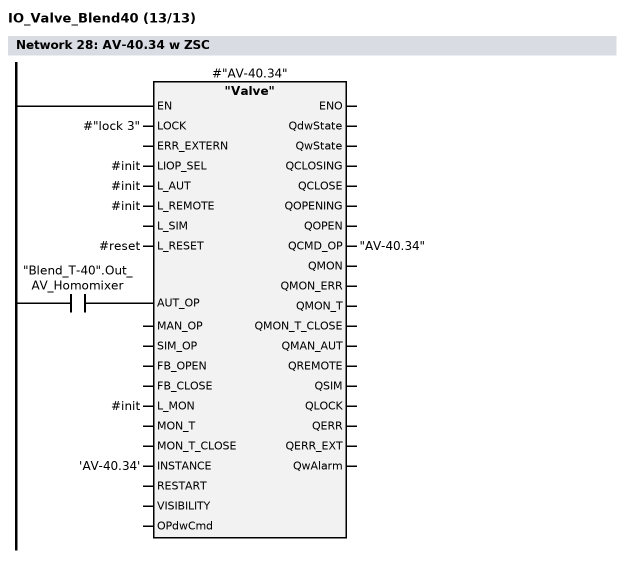
   RUNG wire#powerrail
      #"AV-40.34"(AUT_OP := wire#w1, LOCK := #"lock 3", ERR_EXTERN :=, LIOP_SEL := #init, L_AUT := #init, L_REMOTE := #init, L_SIM :=, L_RESET := #reset, MAN_OP :=, SIM_OP :=, FB_OPEN :=, FB_CLOSE :=, L_MON := #init, MON_T :=, MON_T_CLOSE :=, INSTANCE := 'AV-40.34', RESTART :=, VISIBILITY :=, OPdwCmd :=, QdwState =>, QwState =>, QCLOSING =>, QCLOSE =>, QOPENING =>, QOPEN =>, QCMD_OP => "AV-40.34", QMON =>, QMON_ERR =>, QMON_T =>, QMON_T_CLOSE =>, QMAN_AUT =>, QREMOTE =>, QSIM =>, QLOCK =>, QERR =>, QERR_EXT =>, QwAlarm =>)
   END_RUNG
   RUNG wire#powerrail
      Contact( "Blend_T-40".Out_AV_Homomixer )
   END_RUNG wire#w1
   // the same network as SCL:
   #"AV-40.34"(LOCK := #"lock 3",   // "Valve"
               LIOP_SEL := #init,
               L_AUT := #init,
               L_REMOTE := #init,
               L_RESET := #reset,
               AUT_OP := "Blend_T-40".Out_AV_Homomixer,
               L_MON := #init,
               INSTANCE := 'AV-40.34',
               QCMD_OP => "AV-40.34");
END_REGION
END_FUNCTION_BLOCK

FUNCTION_BLOCK "IO_Valve_Blend41"   // FB29, LAD
{ S7_Optimized_Access := 'FALSE' }
VERSION : 0.1
// stored: AutoNumber true, IsIECCheckEnabled false, SetENOAutomatically false, UDAEnableTagReadback false
   VAR_INPUT
      "lock 1" : Bool;
      "lock 2" : Bool;
      "lock 3" : Bool;
      "lock 4" : Bool;
      init : Bool;
      reset : Bool;
      testing : Bool;
   END_VAR
   VAR
      "AV-41.01" : "Valve";
      "AV-41.02" : "Valve";
      "AV-41.03" : "Valve";
      "AV-41.04" : "Valve";
      "AV-41.05" : "Valve";
      "AV-41.06" : "Valve";
      "AV-41.07" : "Valve";
      "AV-41.08" : "Valve";
      "AV-41.09" : "Valve";
      "AV-41.10" : "Valve";
      "AV-41.11" : "Valve";
      "AV-41.12" : "Valve";
      "AV-41.13" : "Valve";
      "AV-41.14" : "Valve";
      "AV-41.15" : "Valve";
      "AV-41.16" : "Valve";
      "AV-41.17" : "Valve";
      "AV-41.18" : "Valve";
      "AV-41.19" : "Valve";
      "AV-41.20" : "Valve";
      "AV-41.21" : "Valve";
      "AV-41.22" : "Valve";
      "AV-41.23" : "Valve";
      "AV-41.24" : "Valve";
      "AV-41.25" : "Valve";
      "AV-41.26" : "Valve";
      "AV-41.27" : "Valve";
      "AV-41.28" : "Valve";
      "AV-41.29" : "Valve";
      "AV-41.30" : "Valve";
      "AV-41.31" : "Valve";
      "AV-41.32" : "Valve";
      "AV-41.33" : "Valve";
      "AV-41.34" : "Valve";
   END_VAR
BEGIN

REGION Network 2 (SCL): FB OPEN AND CLOSE VALVE T-41
   IF #testing THEN
       // Statement section IF
       #"AV-41.01".FB_OPEN := #"AV-41.01".QCMD_OP;
       #"AV-41.01".FB_CLOSE := NOT #"AV-41.01".QCMD_OP;
       #"AV-41.02".FB_OPEN := #"AV-41.02".QCMD_OP;
       #"AV-41.02".FB_CLOSE := NOT #"AV-41.02".QCMD_OP;
       #"AV-41.03".FB_OPEN := #"AV-41.03".QCMD_OP;
       #"AV-41.03".FB_CLOSE := NOT #"AV-41.03".QCMD_OP;
       #"AV-41.04".FB_OPEN := #"AV-41.04".QCMD_OP;
       #"AV-41.04".FB_CLOSE := NOT #"AV-41.04".QCMD_OP;
       #"AV-41.05".FB_OPEN := #"AV-41.05".QCMD_OP;
       #"AV-41.05".FB_CLOSE := NOT #"AV-41.05".QCMD_OP;
       #"AV-41.06".FB_OPEN := #"AV-41.06".QCMD_OP;
       #"AV-41.06".FB_CLOSE := NOT #"AV-41.06".QCMD_OP;
       #"AV-41.07".FB_OPEN := #"AV-41.07".QCMD_OP;
       #"AV-41.07".FB_CLOSE := NOT #"AV-41.07".QCMD_OP;
       #"AV-41.08".FB_OPEN := #"AV-41.08".QCMD_OP;
       #"AV-41.08".FB_CLOSE := NOT #"AV-41.08".QCMD_OP;
       #"AV-41.09".FB_OPEN := #"AV-41.09".QCMD_OP;
       #"AV-41.09".FB_CLOSE := NOT #"AV-41.09".QCMD_OP;
       #"AV-41.10".FB_OPEN := #"AV-41.10".QCMD_OP;
       #"AV-41.10".FB_CLOSE := NOT #"AV-41.10".QCMD_OP;
       #"AV-41.11".FB_OPEN := #"AV-41.11".QCMD_OP;
       #"AV-41.11".FB_CLOSE := NOT #"AV-41.11".QCMD_OP;
       #"AV-41.12".FB_OPEN := #"AV-41.12".QCMD_OP;
       #"AV-41.12".FB_CLOSE := NOT #"AV-41.12".QCMD_OP;
       #"AV-41.13".FB_OPEN := #"AV-41.13".QCMD_OP;
       #"AV-41.13".FB_CLOSE := NOT #"AV-41.13".QCMD_OP;
       #"AV-41.14".FB_OPEN := #"AV-41.14".QCMD_OP;
       #"AV-41.14".FB_CLOSE := NOT #"AV-41.14".QCMD_OP;
       #"AV-41.15".FB_OPEN := #"AV-41.15".QCMD_OP;
       #"AV-41.15".FB_CLOSE := NOT #"AV-41.15".QCMD_OP;
       #"AV-41.16".FB_OPEN := #"AV-41.16".QCMD_OP;
       #"AV-41.16".FB_CLOSE := NOT #"AV-41.16".QCMD_OP;
       #"AV-41.17".FB_OPEN := #"AV-41.17".QCMD_OP;
       #"AV-41.17".FB_CLOSE := NOT #"AV-41.17".QCMD_OP;
       #"AV-41.18".FB_OPEN := #"AV-41.18".QCMD_OP;
       #"AV-41.18".FB_CLOSE := NOT #"AV-41.18".QCMD_OP;
       #"AV-41.19".FB_OPEN := #"AV-41.19".QCMD_OP;
       #"AV-41.19".FB_CLOSE := NOT #"AV-41.19".QCMD_OP;
       #"AV-41.20".FB_OPEN := #"AV-41.20".QCMD_OP;
       #"AV-41.20".FB_CLOSE := NOT #"AV-41.20".QCMD_OP;
       #"AV-41.21".FB_OPEN := #"AV-41.21".QCMD_OP;
       #"AV-41.21".FB_CLOSE := NOT #"AV-41.21".QCMD_OP;
       #"AV-41.22".FB_OPEN := #"AV-41.22".QCMD_OP;
       #"AV-41.22".FB_CLOSE := NOT #"AV-41.22".QCMD_OP;
       #"AV-41.23".FB_OPEN := #"AV-41.23".QCMD_OP;
       #"AV-41.23".FB_CLOSE := NOT #"AV-41.23".QCMD_OP;
       #"AV-41.24".FB_OPEN := #"AV-41.24".QCMD_OP;
       #"AV-41.24".FB_CLOSE := NOT #"AV-41.24".QCMD_OP;
       #"AV-41.25".FB_OPEN := #"AV-41.25".QCMD_OP;
       #"AV-41.25".FB_CLOSE := NOT #"AV-41.25".QCMD_OP;
       #"AV-41.26".FB_OPEN := #"AV-41.26".QCMD_OP;
       #"AV-41.26".FB_CLOSE := NOT #"AV-41.26".QCMD_OP;
       #"AV-41.27".FB_OPEN := #"AV-41.27".QCMD_OP;
       #"AV-41.27".FB_CLOSE := NOT #"AV-41.27".QCMD_OP;
       #"AV-41.28".FB_OPEN := #"AV-41.28".QCMD_OP;
       #"AV-41.28".FB_CLOSE := NOT #"AV-41.28".QCMD_OP;
       #"AV-41.29".FB_OPEN := #"AV-41.29".QCMD_OP;
       #"AV-41.29".FB_CLOSE := NOT #"AV-41.29".QCMD_OP;
       #"AV-41.30".FB_OPEN := #"AV-41.30".QCMD_OP;
       #"AV-41.30".FB_CLOSE := NOT #"AV-41.30".QCMD_OP;
       #"AV-41.31".FB_OPEN := #"AV-41.31".QCMD_OP;
       #"AV-41.31".FB_CLOSE := NOT #"AV-41.31".QCMD_OP;
       #"AV-41.32".FB_OPEN := #"AV-41.32".QCMD_OP;
       #"AV-41.32".FB_CLOSE := NOT #"AV-41.32".QCMD_OP;
       #"AV-41.33".FB_OPEN := #"AV-41.33".QCMD_OP;
       #"AV-41.33".FB_CLOSE := NOT #"AV-41.33".QCMD_OP;
       #"AV-41.34".FB_OPEN := #"AV-41.34".QCMD_OP;
       #"AV-41.34".FB_CLOSE := NOT #"AV-41.34".QCMD_OP;
   ELSE
       // Statement section ELSE
       #"AV-41.01".FB_OPEN := #"AV-41.01".QCMD_OP;
       #"AV-41.01".FB_CLOSE := NOT #"AV-41.01".QCMD_OP;
       #"AV-41.02".FB_OPEN := NOT "ZSC-41.02";
       #"AV-41.02".FB_CLOSE := "ZSC-41.02";
       #"AV-41.03".FB_OPEN := NOT "ZSC-41.03";
       #"AV-41.03".FB_CLOSE := "ZSC-41.03";
       #"AV-41.04".FB_OPEN := #"AV-41.04".QCMD_OP;
       #"AV-41.04".FB_CLOSE := NOT #"AV-41.04".QCMD_OP;
       #"AV-41.05".FB_OPEN := NOT "ZSC-41.05";
       #"AV-41.05".FB_CLOSE := "ZSC-41.05";
       #"AV-41.06".FB_OPEN := NOT "ZSC-41.06";
       #"AV-41.06".FB_CLOSE := "ZSC-41.06";
       #"AV-41.07".FB_OPEN := #"AV-41.07".QCMD_OP;
       #"AV-41.07".FB_CLOSE := NOT #"AV-41.07".QCMD_OP;
       #"AV-41.08".FB_OPEN := NOT "ZSC-41.08";
       #"AV-41.08".FB_CLOSE := "ZSC-41.08";
       #"AV-41.09".FB_OPEN := NOT "ZSC-41.09";
       #"AV-41.09".FB_CLOSE := "ZSC-41.09";
       #"AV-41.10".FB_OPEN := #"AV-41.10".QCMD_OP;
       #"AV-41.10".FB_CLOSE := NOT #"AV-41.10".QCMD_OP;
       #"AV-41.11".FB_OPEN := NOT "ZSC-41.11";
       #"AV-41.11".FB_CLOSE := "ZSC-41.11";
       #"AV-41.12".FB_OPEN := #"AV-41.12".QCMD_OP;
       #"AV-41.12".FB_CLOSE := NOT #"AV-41.12".QCMD_OP;
       #"AV-41.13".FB_OPEN := #"AV-41.13".QCMD_OP;
       #"AV-41.13".FB_CLOSE := NOT #"AV-41.13".QCMD_OP;
       #"AV-41.14".FB_OPEN := NOT "ZSC-41.14";
       #"AV-41.14".FB_CLOSE := "ZSC-41.14";
       #"AV-41.15".FB_OPEN := #"AV-41.15".QCMD_OP;
       #"AV-41.15".FB_CLOSE := NOT #"AV-41.15".QCMD_OP;
       #"AV-41.16".FB_OPEN := #"AV-41.16".QCMD_OP;
       #"AV-41.16".FB_CLOSE := NOT #"AV-41.16".QCMD_OP;
       #"AV-41.17".FB_OPEN := NOT "ZSC-41.17";
       #"AV-41.17".FB_CLOSE := "ZSC-41.17";
       #"AV-41.18".FB_OPEN := #"AV-41.18".QCMD_OP;
       #"AV-41.18".FB_CLOSE := NOT #"AV-41.18".QCMD_OP;
       #"AV-41.19".FB_OPEN := #"AV-41.19".QCMD_OP;
       #"AV-41.19".FB_CLOSE := NOT #"AV-41.19".QCMD_OP;
       #"AV-41.20".FB_OPEN := NOT "ZSC-41.20";
       #"AV-41.20".FB_CLOSE := "ZSC-41.20";
       #"AV-41.21".FB_OPEN := NOT "ZSC-41.21";
       #"AV-41.21".FB_CLOSE := "ZSC-41.21";
       #"AV-41.22".FB_OPEN := #"AV-41.22".QCMD_OP;
       #"AV-41.22".FB_CLOSE := NOT #"AV-41.22".QCMD_OP;
       #"AV-41.23".FB_OPEN := NOT "ZSC-41.23";
       #"AV-41.23".FB_CLOSE := "ZSC-41.23";
       #"AV-41.24".FB_OPEN := NOT "ZSC-41.24";
       #"AV-41.24".FB_CLOSE := "ZSC-41.24";
       #"AV-41.25".FB_OPEN := NOT "ZSC-41.25";
       #"AV-41.25".FB_CLOSE := "ZSC-41.25";
       #"AV-41.26".FB_OPEN := #"AV-41.26".QCMD_OP;
       #"AV-41.26".FB_CLOSE := NOT #"AV-41.26".QCMD_OP;
       #"AV-41.27".FB_OPEN := NOT "ZSC-41.27";
       #"AV-41.27".FB_CLOSE := "ZSC-41.27";
       #"AV-41.28".FB_OPEN := NOT "ZSC-41.28";
       #"AV-41.28".FB_CLOSE := "ZSC-41.28";
       #"AV-41.29".FB_OPEN := #"AV-41.29".QCMD_OP;
       #"AV-41.29".FB_CLOSE := NOT #"AV-41.29".QCMD_OP;
       #"AV-41.30".FB_OPEN := #"AV-41.30".QCMD_OP;
       #"AV-41.30".FB_CLOSE := NOT #"AV-41.30".QCMD_OP;
       #"AV-41.31".FB_OPEN := NOT "ZSC-41.31";
       #"AV-41.31".FB_CLOSE := "ZSC-41.31";
       #"AV-41.32".FB_OPEN := NOT "ZSC-41.32";
       #"AV-41.32".FB_CLOSE := "ZSC-41.32";
       #"AV-41.33".FB_OPEN := NOT "ZSC-41.33";
       #"AV-41.33".FB_CLOSE := "ZSC-41.33";
       #"AV-41.34".FB_OPEN := NOT "ZSC-41.34";
       #"AV-41.34".FB_CLOSE := "ZSC-41.34";
   END_IF;
END_REGION

NETWORK
TITLE = FB MONITORING TIME VALVE T-41
// FB OPEN TIME
      L     T#20s;
      T     #"AV-41.01".MON_T;
      T     #"AV-41.02".MON_T;
      T     #"AV-41.03".MON_T;
      T     #"AV-41.04".MON_T;
      T     #"AV-41.05".MON_T;
      T     #"AV-41.06".MON_T;
      T     #"AV-41.07".MON_T;
      T     #"AV-41.08".MON_T;
      T     #"AV-41.09".MON_T;
      T     #"AV-41.10".MON_T;
      T     #"AV-41.11".MON_T;
      T     #"AV-41.12".MON_T;
      T     #"AV-41.13".MON_T;
      T     #"AV-41.14".MON_T;
      T     #"AV-41.15".MON_T;
      T     #"AV-41.16".MON_T;
      T     #"AV-41.17".MON_T;
      T     #"AV-41.18".MON_T;
      T     #"AV-41.19".MON_T;
      T     #"AV-41.20".MON_T;
      T     #"AV-41.21".MON_T;
      T     #"AV-41.22".MON_T;
      T     #"AV-41.23".MON_T;
      T     #"AV-41.24".MON_T;
      T     #"AV-41.25".MON_T;
      T     #"AV-41.26".MON_T;
      T     #"AV-41.27".MON_T;
      T     #"AV-41.28".MON_T;
      T     #"AV-41.29".MON_T;
      T     #"AV-41.30".MON_T;
      T     #"AV-41.31".MON_T;
      T     #"AV-41.32".MON_T;
      T     #"AV-41.33".MON_T;
      T     #"AV-41.34".MON_T;
// FB CLOSE TIME
      L     T#20s;
      T     #"AV-41.01".MON_T_CLOSE;
      T     #"AV-41.02".MON_T_CLOSE;
      T     #"AV-41.03".MON_T_CLOSE;
      T     #"AV-41.04".MON_T_CLOSE;
      T     #"AV-41.05".MON_T_CLOSE;
      T     #"AV-41.06".MON_T_CLOSE;
      T     #"AV-41.07".MON_T_CLOSE;
      T     #"AV-41.08".MON_T_CLOSE;
      T     #"AV-41.09".MON_T_CLOSE;
      T     #"AV-41.10".MON_T_CLOSE;
      T     #"AV-41.11".MON_T_CLOSE;
      T     #"AV-41.12".MON_T_CLOSE;
      T     #"AV-41.13".MON_T_CLOSE;
      T     #"AV-41.14".MON_T_CLOSE;
      T     #"AV-41.15".MON_T_CLOSE;
      T     #"AV-41.16".MON_T_CLOSE;
      T     #"AV-41.17".MON_T_CLOSE;
      T     #"AV-41.18".MON_T_CLOSE;
      T     #"AV-41.19".MON_T_CLOSE;
      T     #"AV-41.20".MON_T_CLOSE;
      T     #"AV-41.21".MON_T_CLOSE;
      T     #"AV-41.22".MON_T_CLOSE;
      T     #"AV-41.23".MON_T_CLOSE;
      T     #"AV-41.24".MON_T_CLOSE;
      T     #"AV-41.25".MON_T_CLOSE;
      T     #"AV-41.26".MON_T_CLOSE;
      T     #"AV-41.27".MON_T_CLOSE;
      T     #"AV-41.28".MON_T_CLOSE;
      T     #"AV-41.29".MON_T_CLOSE;
      T     #"AV-41.30".MON_T_CLOSE;
      T     #"AV-41.31".MON_T_CLOSE;
      T     #"AV-41.32".MON_T_CLOSE;
      T     #"AV-41.33".MON_T_CLOSE;
      T     #"AV-41.34".MON_T_CLOSE;

REGION Network 4: AV-41.01
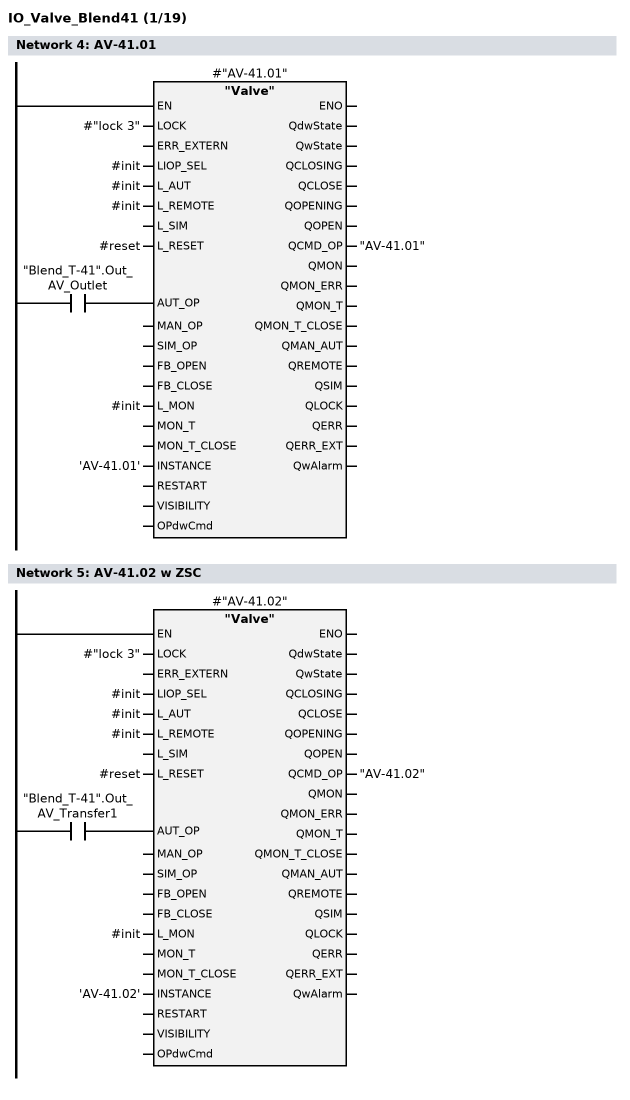
   RUNG wire#powerrail
      #"AV-41.01"(AUT_OP := wire#w1, LOCK := #"lock 3", ERR_EXTERN :=, LIOP_SEL := #init, L_AUT := #init, L_REMOTE := #init, L_SIM :=, L_RESET := #reset, MAN_OP :=, SIM_OP :=, FB_OPEN :=, FB_CLOSE :=, L_MON := #init, MON_T :=, MON_T_CLOSE :=, INSTANCE := 'AV-41.01', RESTART :=, VISIBILITY :=, OPdwCmd :=, QdwState =>, QwState =>, QCLOSING =>, QCLOSE =>, QOPENING =>, QOPEN =>, QCMD_OP => "AV-41.01", QMON =>, QMON_ERR =>, QMON_T =>, QMON_T_CLOSE =>, QMAN_AUT =>, QREMOTE =>, QSIM =>, QLOCK =>, QERR =>, QERR_EXT =>, QwAlarm =>)
   END_RUNG
   RUNG wire#powerrail
      Contact( "Blend_T-41".Out_AV_Outlet )
   END_RUNG wire#w1
   // the same network as SCL:
   #"AV-41.01"(LOCK := #"lock 3",   // "Valve"
               LIOP_SEL := #init,
               L_AUT := #init,
               L_REMOTE := #init,
               L_RESET := #reset,
               AUT_OP := "Blend_T-41".Out_AV_Outlet,
               L_MON := #init,
               INSTANCE := 'AV-41.01',
               QCMD_OP => "AV-41.01");
END_REGION

REGION Network 5: AV-41.02 w ZSC
   RUNG wire#powerrail
      #"AV-41.02"(AUT_OP := wire#w1, LOCK := #"lock 3", ERR_EXTERN :=, LIOP_SEL := #init, L_AUT := #init, L_REMOTE := #init, L_SIM :=, L_RESET := #reset, MAN_OP :=, SIM_OP :=, FB_OPEN :=, FB_CLOSE :=, L_MON := #init, MON_T :=, MON_T_CLOSE :=, INSTANCE := 'AV-41.02', RESTART :=, VISIBILITY :=, OPdwCmd :=, QdwState =>, QwState =>, QCLOSING =>, QCLOSE =>, QOPENING =>, QOPEN =>, QCMD_OP => "AV-41.02", QMON =>, QMON_ERR =>, QMON_T =>, QMON_T_CLOSE =>, QMAN_AUT =>, QREMOTE =>, QSIM =>, QLOCK =>, QERR =>, QERR_EXT =>, QwAlarm =>)
   END_RUNG
   RUNG wire#powerrail
      Contact( "Blend_T-41".Out_AV_Transfer1 )
   END_RUNG wire#w1
   // the same network as SCL:
   #"AV-41.02"(LOCK := #"lock 3",   // "Valve"
               LIOP_SEL := #init,
               L_AUT := #init,
               L_REMOTE := #init,
               L_RESET := #reset,
               AUT_OP := "Blend_T-41".Out_AV_Transfer1,
               L_MON := #init,
               INSTANCE := 'AV-41.02',
               QCMD_OP => "AV-41.02");
END_REGION

REGION Network 6: AV-41.03 w ZSC
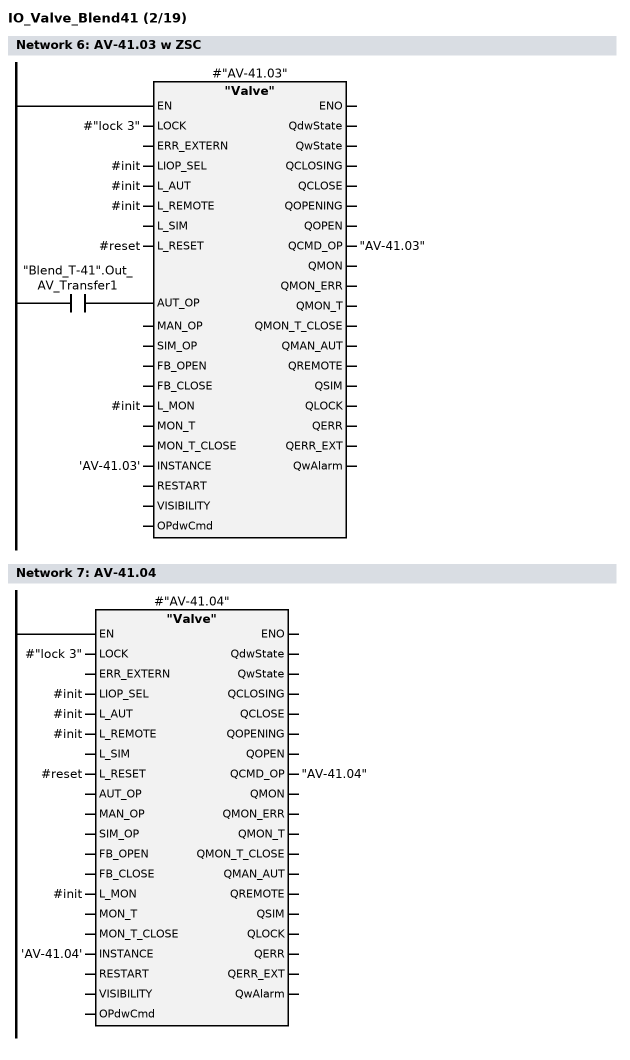
   RUNG wire#powerrail
      #"AV-41.03"(AUT_OP := wire#w1, LOCK := #"lock 3", ERR_EXTERN :=, LIOP_SEL := #init, L_AUT := #init, L_REMOTE := #init, L_SIM :=, L_RESET := #reset, MAN_OP :=, SIM_OP :=, FB_OPEN :=, FB_CLOSE :=, L_MON := #init, MON_T :=, MON_T_CLOSE :=, INSTANCE := 'AV-41.03', RESTART :=, VISIBILITY :=, OPdwCmd :=, QdwState =>, QwState =>, QCLOSING =>, QCLOSE =>, QOPENING =>, QOPEN =>, QCMD_OP => "AV-41.03", QMON =>, QMON_ERR =>, QMON_T =>, QMON_T_CLOSE =>, QMAN_AUT =>, QREMOTE =>, QSIM =>, QLOCK =>, QERR =>, QERR_EXT =>, QwAlarm =>)
   END_RUNG
   RUNG wire#powerrail
      Contact( "Blend_T-41".Out_AV_Transfer1 )
   END_RUNG wire#w1
   // the same network as SCL:
   #"AV-41.03"(LOCK := #"lock 3",   // "Valve"
               LIOP_SEL := #init,
               L_AUT := #init,
               L_REMOTE := #init,
               L_RESET := #reset,
               AUT_OP := "Blend_T-41".Out_AV_Transfer1,
               L_MON := #init,
               INSTANCE := 'AV-41.03',
               QCMD_OP => "AV-41.03");
END_REGION

REGION Network 7: AV-41.04
   RUNG wire#powerrail
      #"AV-41.04"(LOCK := #"lock 3", ERR_EXTERN :=, LIOP_SEL := #init, L_AUT := #init, L_REMOTE := #init, L_SIM :=, L_RESET := #reset, AUT_OP :=, MAN_OP :=, SIM_OP :=, FB_OPEN :=, FB_CLOSE :=, L_MON := #init, MON_T :=, MON_T_CLOSE :=, INSTANCE := 'AV-41.04', RESTART :=, VISIBILITY :=, OPdwCmd :=, QdwState =>, QwState =>, QCLOSING =>, QCLOSE =>, QOPENING =>, QOPEN =>, QCMD_OP => "AV-41.04", QMON =>, QMON_ERR =>, QMON_T =>, QMON_T_CLOSE =>, QMAN_AUT =>, QREMOTE =>, QSIM =>, QLOCK =>, QERR =>, QERR_EXT =>, QwAlarm =>)
   END_RUNG
   // the same network as SCL:
   #"AV-41.04"(LOCK := #"lock 3",   // "Valve"
               LIOP_SEL := #init,
               L_AUT := #init,
               L_REMOTE := #init,
               L_RESET := #reset,
               L_MON := #init,
               INSTANCE := 'AV-41.04',
               QCMD_OP => "AV-41.04");
END_REGION

REGION Network 8: AV-41.05 w ZSC
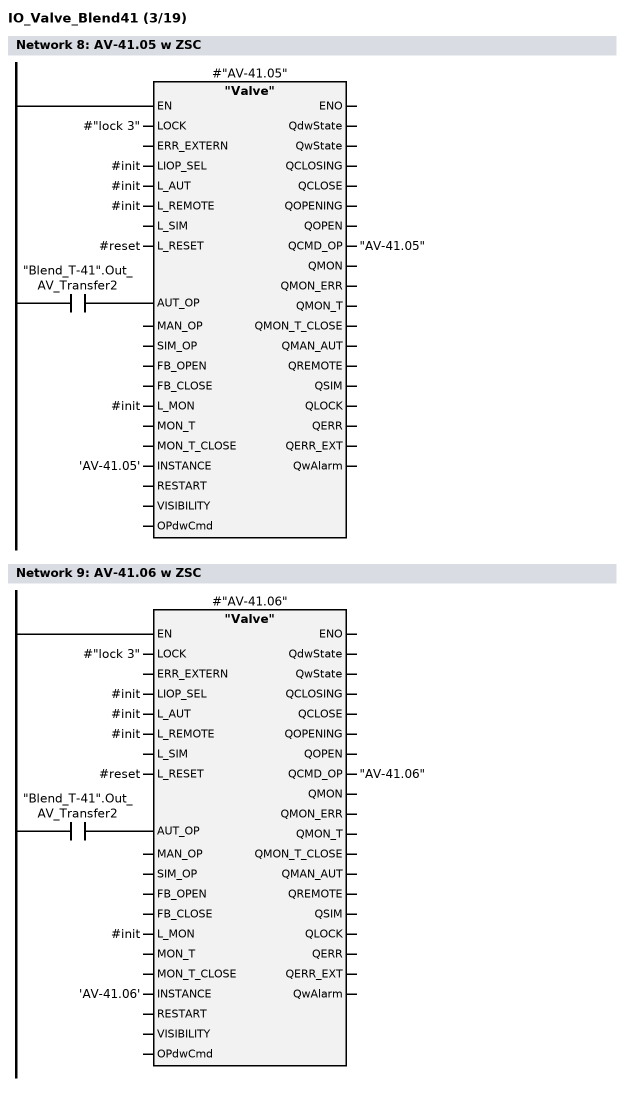
   RUNG wire#powerrail
      #"AV-41.05"(AUT_OP := wire#w1, LOCK := #"lock 3", ERR_EXTERN :=, LIOP_SEL := #init, L_AUT := #init, L_REMOTE := #init, L_SIM :=, L_RESET := #reset, MAN_OP :=, SIM_OP :=, FB_OPEN :=, FB_CLOSE :=, L_MON := #init, MON_T :=, MON_T_CLOSE :=, INSTANCE := 'AV-41.05', RESTART :=, VISIBILITY :=, OPdwCmd :=, QdwState =>, QwState =>, QCLOSING =>, QCLOSE =>, QOPENING =>, QOPEN =>, QCMD_OP => "AV-41.05", QMON =>, QMON_ERR =>, QMON_T =>, QMON_T_CLOSE =>, QMAN_AUT =>, QREMOTE =>, QSIM =>, QLOCK =>, QERR =>, QERR_EXT =>, QwAlarm =>)
   END_RUNG
   RUNG wire#powerrail
      Contact( "Blend_T-41".Out_AV_Transfer2 )
   END_RUNG wire#w1
   // the same network as SCL:
   #"AV-41.05"(LOCK := #"lock 3",   // "Valve"
               LIOP_SEL := #init,
               L_AUT := #init,
               L_REMOTE := #init,
               L_RESET := #reset,
               AUT_OP := "Blend_T-41".Out_AV_Transfer2,
               L_MON := #init,
               INSTANCE := 'AV-41.05',
               QCMD_OP => "AV-41.05");
END_REGION

REGION Network 9: AV-41.06 w ZSC
   RUNG wire#powerrail
      #"AV-41.06"(AUT_OP := wire#w1, LOCK := #"lock 3", ERR_EXTERN :=, LIOP_SEL := #init, L_AUT := #init, L_REMOTE := #init, L_SIM :=, L_RESET := #reset, MAN_OP :=, SIM_OP :=, FB_OPEN :=, FB_CLOSE :=, L_MON := #init, MON_T :=, MON_T_CLOSE :=, INSTANCE := 'AV-41.06', RESTART :=, VISIBILITY :=, OPdwCmd :=, QdwState =>, QwState =>, QCLOSING =>, QCLOSE =>, QOPENING =>, QOPEN =>, QCMD_OP => "AV-41.06", QMON =>, QMON_ERR =>, QMON_T =>, QMON_T_CLOSE =>, QMAN_AUT =>, QREMOTE =>, QSIM =>, QLOCK =>, QERR =>, QERR_EXT =>, QwAlarm =>)
   END_RUNG
   RUNG wire#powerrail
      Contact( "Blend_T-41".Out_AV_Transfer2 )
   END_RUNG wire#w1
   // the same network as SCL:
   #"AV-41.06"(LOCK := #"lock 3",   // "Valve"
               LIOP_SEL := #init,
               L_AUT := #init,
               L_REMOTE := #init,
               L_RESET := #reset,
               AUT_OP := "Blend_T-41".Out_AV_Transfer2,
               L_MON := #init,
               INSTANCE := 'AV-41.06',
               QCMD_OP => "AV-41.06");
END_REGION

REGION Network 10: AV-41.07
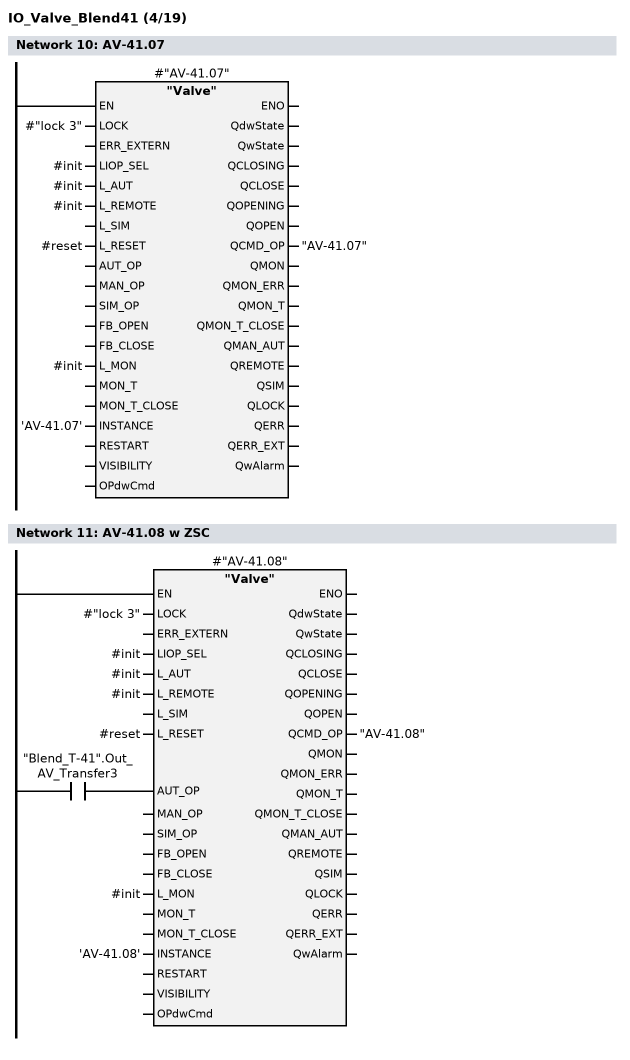
   RUNG wire#powerrail
      #"AV-41.07"(LOCK := #"lock 3", ERR_EXTERN :=, LIOP_SEL := #init, L_AUT := #init, L_REMOTE := #init, L_SIM :=, L_RESET := #reset, AUT_OP :=, MAN_OP :=, SIM_OP :=, FB_OPEN :=, FB_CLOSE :=, L_MON := #init, MON_T :=, MON_T_CLOSE :=, INSTANCE := 'AV-41.07', RESTART :=, VISIBILITY :=, OPdwCmd :=, QdwState =>, QwState =>, QCLOSING =>, QCLOSE =>, QOPENING =>, QOPEN =>, QCMD_OP => "AV-41.07", QMON =>, QMON_ERR =>, QMON_T =>, QMON_T_CLOSE =>, QMAN_AUT =>, QREMOTE =>, QSIM =>, QLOCK =>, QERR =>, QERR_EXT =>, QwAlarm =>)
   END_RUNG
   // the same network as SCL:
   #"AV-41.07"(LOCK := #"lock 3",   // "Valve"
               LIOP_SEL := #init,
               L_AUT := #init,
               L_REMOTE := #init,
               L_RESET := #reset,
               L_MON := #init,
               INSTANCE := 'AV-41.07',
               QCMD_OP => "AV-41.07");
END_REGION

REGION Network 11: AV-41.08 w ZSC
   RUNG wire#powerrail
      #"AV-41.08"(AUT_OP := wire#w1, LOCK := #"lock 3", ERR_EXTERN :=, LIOP_SEL := #init, L_AUT := #init, L_REMOTE := #init, L_SIM :=, L_RESET := #reset, MAN_OP :=, SIM_OP :=, FB_OPEN :=, FB_CLOSE :=, L_MON := #init, MON_T :=, MON_T_CLOSE :=, INSTANCE := 'AV-41.08', RESTART :=, VISIBILITY :=, OPdwCmd :=, QdwState =>, QwState =>, QCLOSING =>, QCLOSE =>, QOPENING =>, QOPEN =>, QCMD_OP => "AV-41.08", QMON =>, QMON_ERR =>, QMON_T =>, QMON_T_CLOSE =>, QMAN_AUT =>, QREMOTE =>, QSIM =>, QLOCK =>, QERR =>, QERR_EXT =>, QwAlarm =>)
   END_RUNG
   RUNG wire#powerrail
      Contact( "Blend_T-41".Out_AV_Transfer3 )
   END_RUNG wire#w1
   // the same network as SCL:
   #"AV-41.08"(LOCK := #"lock 3",   // "Valve"
               LIOP_SEL := #init,
               L_AUT := #init,
               L_REMOTE := #init,
               L_RESET := #reset,
               AUT_OP := "Blend_T-41".Out_AV_Transfer3,
               L_MON := #init,
               INSTANCE := 'AV-41.08',
               QCMD_OP => "AV-41.08");
END_REGION

REGION Network 12: AV-41.09 w ZSC
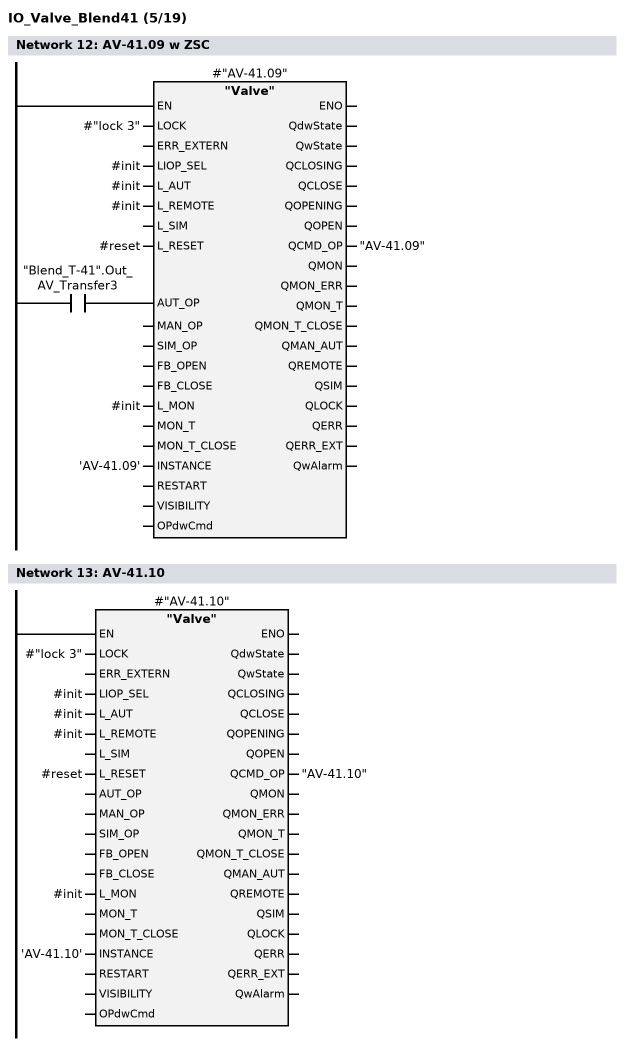
   RUNG wire#powerrail
      #"AV-41.09"(AUT_OP := wire#w1, LOCK := #"lock 3", ERR_EXTERN :=, LIOP_SEL := #init, L_AUT := #init, L_REMOTE := #init, L_SIM :=, L_RESET := #reset, MAN_OP :=, SIM_OP :=, FB_OPEN :=, FB_CLOSE :=, L_MON := #init, MON_T :=, MON_T_CLOSE :=, INSTANCE := 'AV-41.09', RESTART :=, VISIBILITY :=, OPdwCmd :=, QdwState =>, QwState =>, QCLOSING =>, QCLOSE =>, QOPENING =>, QOPEN =>, QCMD_OP => "AV-41.09", QMON =>, QMON_ERR =>, QMON_T =>, QMON_T_CLOSE =>, QMAN_AUT =>, QREMOTE =>, QSIM =>, QLOCK =>, QERR =>, QERR_EXT =>, QwAlarm =>)
   END_RUNG
   RUNG wire#powerrail
      Contact( "Blend_T-41".Out_AV_Transfer3 )
   END_RUNG wire#w1
   // the same network as SCL:
   #"AV-41.09"(LOCK := #"lock 3",   // "Valve"
               LIOP_SEL := #init,
               L_AUT := #init,
               L_REMOTE := #init,
               L_RESET := #reset,
               AUT_OP := "Blend_T-41".Out_AV_Transfer3,
               L_MON := #init,
               INSTANCE := 'AV-41.09',
               QCMD_OP => "AV-41.09");
END_REGION

REGION Network 13: AV-41.10
   RUNG wire#powerrail
      #"AV-41.10"(LOCK := #"lock 3", ERR_EXTERN :=, LIOP_SEL := #init, L_AUT := #init, L_REMOTE := #init, L_SIM :=, L_RESET := #reset, AUT_OP :=, MAN_OP :=, SIM_OP :=, FB_OPEN :=, FB_CLOSE :=, L_MON := #init, MON_T :=, MON_T_CLOSE :=, INSTANCE := 'AV-41.10', RESTART :=, VISIBILITY :=, OPdwCmd :=, QdwState =>, QwState =>, QCLOSING =>, QCLOSE =>, QOPENING =>, QOPEN =>, QCMD_OP => "AV-41.10", QMON =>, QMON_ERR =>, QMON_T =>, QMON_T_CLOSE =>, QMAN_AUT =>, QREMOTE =>, QSIM =>, QLOCK =>, QERR =>, QERR_EXT =>, QwAlarm =>)
   END_RUNG
   // the same network as SCL:
   #"AV-41.10"(LOCK := #"lock 3",   // "Valve"
               LIOP_SEL := #init,
               L_AUT := #init,
               L_REMOTE := #init,
               L_RESET := #reset,
               L_MON := #init,
               INSTANCE := 'AV-41.10',
               QCMD_OP => "AV-41.10");
END_REGION

REGION Network 14: AV-41.11 w ZSC
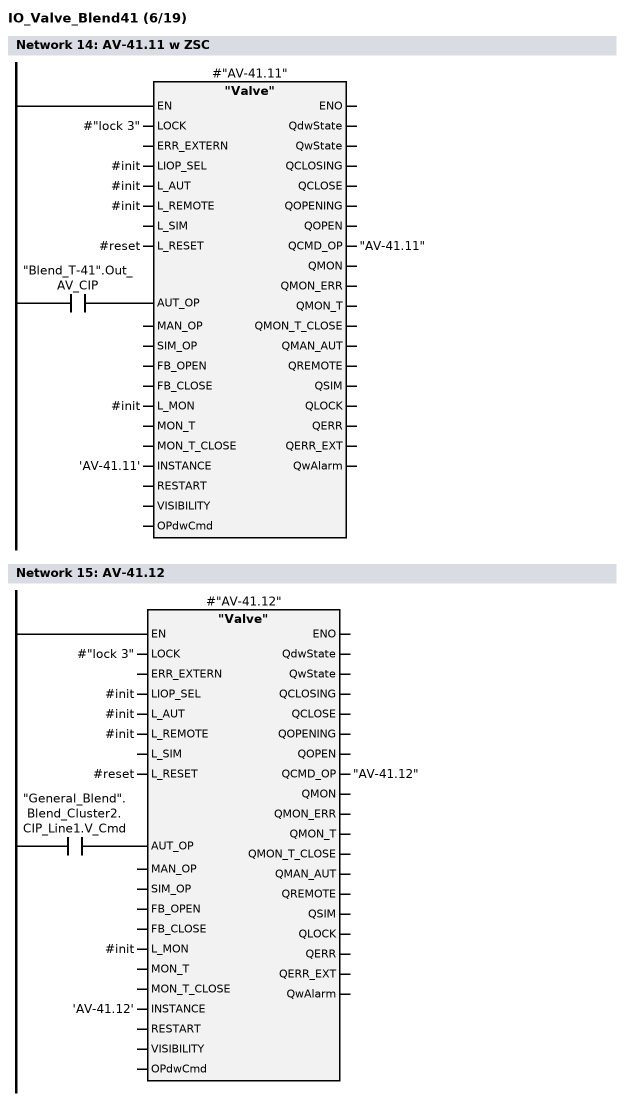
   RUNG wire#powerrail
      #"AV-41.11"(AUT_OP := wire#w1, LOCK := #"lock 3", ERR_EXTERN :=, LIOP_SEL := #init, L_AUT := #init, L_REMOTE := #init, L_SIM :=, L_RESET := #reset, MAN_OP :=, SIM_OP :=, FB_OPEN :=, FB_CLOSE :=, L_MON := #init, MON_T :=, MON_T_CLOSE :=, INSTANCE := 'AV-41.11', RESTART :=, VISIBILITY :=, OPdwCmd :=, QdwState =>, QwState =>, QCLOSING =>, QCLOSE =>, QOPENING =>, QOPEN =>, QCMD_OP => "AV-41.11", QMON =>, QMON_ERR =>, QMON_T =>, QMON_T_CLOSE =>, QMAN_AUT =>, QREMOTE =>, QSIM =>, QLOCK =>, QERR =>, QERR_EXT =>, QwAlarm =>)
   END_RUNG
   RUNG wire#powerrail
      Contact( "Blend_T-41".Out_AV_CIP )
   END_RUNG wire#w1
   // the same network as SCL:
   #"AV-41.11"(LOCK := #"lock 3",   // "Valve"
               LIOP_SEL := #init,
               L_AUT := #init,
               L_REMOTE := #init,
               L_RESET := #reset,
               AUT_OP := "Blend_T-41".Out_AV_CIP,
               L_MON := #init,
               INSTANCE := 'AV-41.11',
               QCMD_OP => "AV-41.11");
END_REGION

REGION Network 15: AV-41.12
   RUNG wire#powerrail
      #"AV-41.12"(AUT_OP := wire#w1, LOCK := #"lock 3", ERR_EXTERN :=, LIOP_SEL := #init, L_AUT := #init, L_REMOTE := #init, L_SIM :=, L_RESET := #reset, MAN_OP :=, SIM_OP :=, FB_OPEN :=, FB_CLOSE :=, L_MON := #init, MON_T :=, MON_T_CLOSE :=, INSTANCE := 'AV-41.12', RESTART :=, VISIBILITY :=, OPdwCmd :=, QdwState =>, QwState =>, QCLOSING =>, QCLOSE =>, QOPENING =>, QOPEN =>, QCMD_OP => "AV-41.12", QMON =>, QMON_ERR =>, QMON_T =>, QMON_T_CLOSE =>, QMAN_AUT =>, QREMOTE =>, QSIM =>, QLOCK =>, QERR =>, QERR_EXT =>, QwAlarm =>)
   END_RUNG
   RUNG wire#powerrail
      Contact( "General_Blend".Blend_Cluster2.CIP_Line1.V_Cmd )
   END_RUNG wire#w1
   // the same network as SCL:
   #"AV-41.12"(LOCK := #"lock 3",   // "Valve"
               LIOP_SEL := #init,
               L_AUT := #init,
               L_REMOTE := #init,
               L_RESET := #reset,
               AUT_OP := "General_Blend".Blend_Cluster2.CIP_Line1.V_Cmd,
               L_MON := #init,
               INSTANCE := 'AV-41.12',
               QCMD_OP => "AV-41.12");
END_REGION

REGION Network 16: AV-41.13
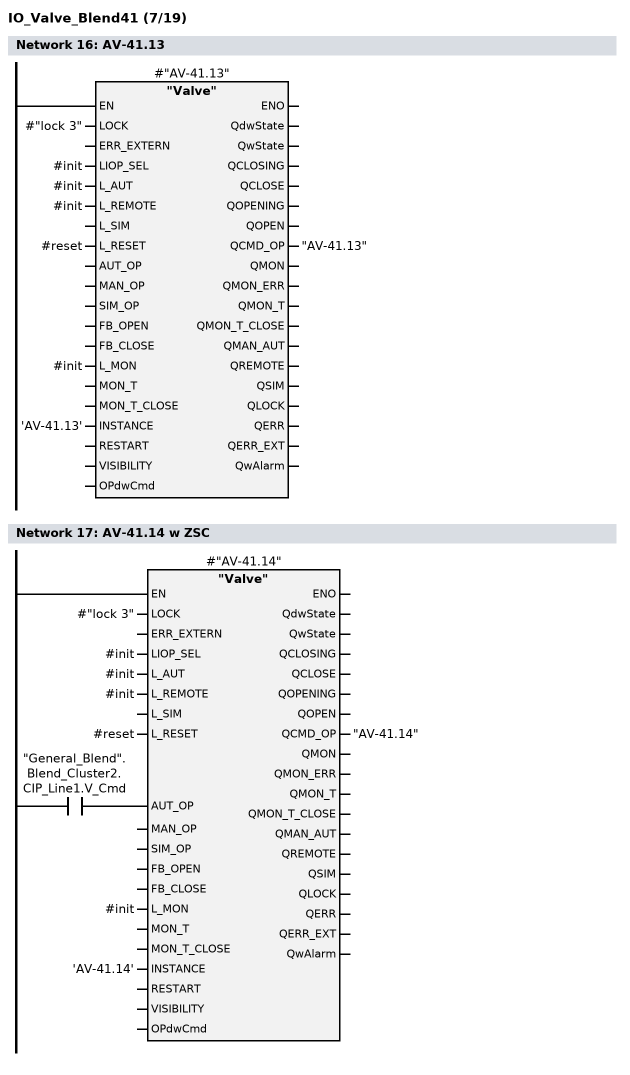
   RUNG wire#powerrail
      #"AV-41.13"(LOCK := #"lock 3", ERR_EXTERN :=, LIOP_SEL := #init, L_AUT := #init, L_REMOTE := #init, L_SIM :=, L_RESET := #reset, AUT_OP :=, MAN_OP :=, SIM_OP :=, FB_OPEN :=, FB_CLOSE :=, L_MON := #init, MON_T :=, MON_T_CLOSE :=, INSTANCE := 'AV-41.13', RESTART :=, VISIBILITY :=, OPdwCmd :=, QdwState =>, QwState =>, QCLOSING =>, QCLOSE =>, QOPENING =>, QOPEN =>, QCMD_OP => "AV-41.13", QMON =>, QMON_ERR =>, QMON_T =>, QMON_T_CLOSE =>, QMAN_AUT =>, QREMOTE =>, QSIM =>, QLOCK =>, QERR =>, QERR_EXT =>, QwAlarm =>)
   END_RUNG
   // the same network as SCL:
   #"AV-41.13"(LOCK := #"lock 3",   // "Valve"
               LIOP_SEL := #init,
               L_AUT := #init,
               L_REMOTE := #init,
               L_RESET := #reset,
               L_MON := #init,
               INSTANCE := 'AV-41.13',
               QCMD_OP => "AV-41.13");
END_REGION

REGION Network 17: AV-41.14 w ZSC
   RUNG wire#powerrail
      #"AV-41.14"(AUT_OP := wire#w1, LOCK := #"lock 3", ERR_EXTERN :=, LIOP_SEL := #init, L_AUT := #init, L_REMOTE := #init, L_SIM :=, L_RESET := #reset, MAN_OP :=, SIM_OP :=, FB_OPEN :=, FB_CLOSE :=, L_MON := #init, MON_T :=, MON_T_CLOSE :=, INSTANCE := 'AV-41.14', RESTART :=, VISIBILITY :=, OPdwCmd :=, QdwState =>, QwState =>, QCLOSING =>, QCLOSE =>, QOPENING =>, QOPEN =>, QCMD_OP => "AV-41.14", QMON =>, QMON_ERR =>, QMON_T =>, QMON_T_CLOSE =>, QMAN_AUT =>, QREMOTE =>, QSIM =>, QLOCK =>, QERR =>, QERR_EXT =>, QwAlarm =>)
   END_RUNG
   RUNG wire#powerrail
      Contact( "General_Blend".Blend_Cluster2.CIP_Line1.V_Cmd )
   END_RUNG wire#w1
   // the same network as SCL:
   #"AV-41.14"(LOCK := #"lock 3",   // "Valve"
               LIOP_SEL := #init,
               L_AUT := #init,
               L_REMOTE := #init,
               L_RESET := #reset,
               AUT_OP := "General_Blend".Blend_Cluster2.CIP_Line1.V_Cmd,
               L_MON := #init,
               INSTANCE := 'AV-41.14',
               QCMD_OP => "AV-41.14");
END_REGION

REGION Network 18: AV-41.15
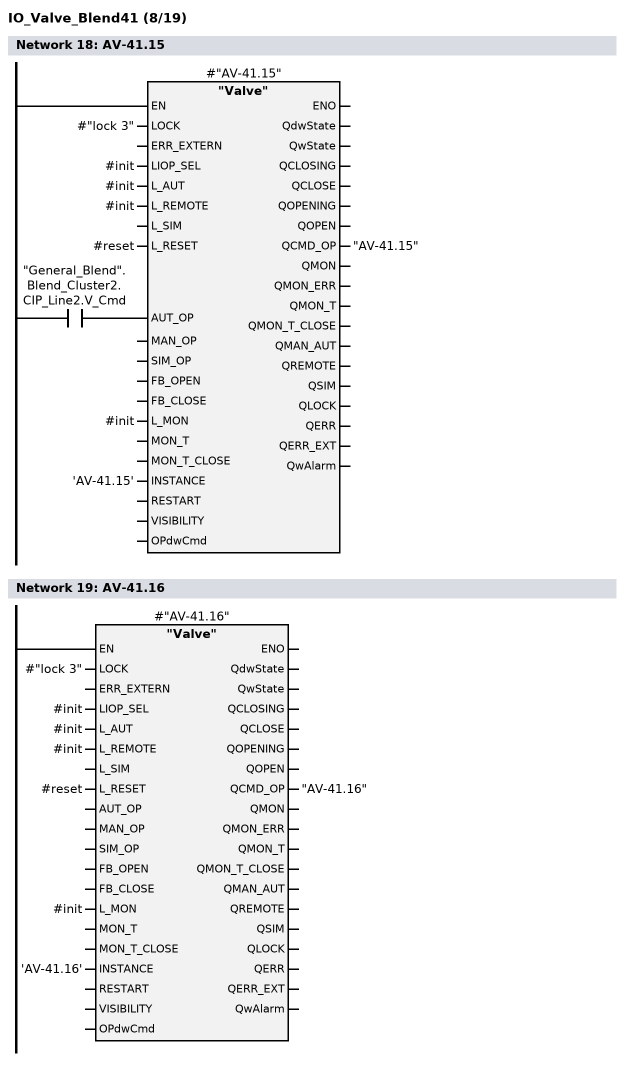
   RUNG wire#powerrail
      #"AV-41.15"(AUT_OP := wire#w1, LOCK := #"lock 3", ERR_EXTERN :=, LIOP_SEL := #init, L_AUT := #init, L_REMOTE := #init, L_SIM :=, L_RESET := #reset, MAN_OP :=, SIM_OP :=, FB_OPEN :=, FB_CLOSE :=, L_MON := #init, MON_T :=, MON_T_CLOSE :=, INSTANCE := 'AV-41.15', RESTART :=, VISIBILITY :=, OPdwCmd :=, QdwState =>, QwState =>, QCLOSING =>, QCLOSE =>, QOPENING =>, QOPEN =>, QCMD_OP => "AV-41.15", QMON =>, QMON_ERR =>, QMON_T =>, QMON_T_CLOSE =>, QMAN_AUT =>, QREMOTE =>, QSIM =>, QLOCK =>, QERR =>, QERR_EXT =>, QwAlarm =>)
   END_RUNG
   RUNG wire#powerrail
      Contact( "General_Blend".Blend_Cluster2.CIP_Line2.V_Cmd )
   END_RUNG wire#w1
   // the same network as SCL:
   #"AV-41.15"(LOCK := #"lock 3",   // "Valve"
               LIOP_SEL := #init,
               L_AUT := #init,
               L_REMOTE := #init,
               L_RESET := #reset,
               AUT_OP := "General_Blend".Blend_Cluster2.CIP_Line2.V_Cmd,
               L_MON := #init,
               INSTANCE := 'AV-41.15',
               QCMD_OP => "AV-41.15");
END_REGION

REGION Network 19: AV-41.16
   RUNG wire#powerrail
      #"AV-41.16"(LOCK := #"lock 3", ERR_EXTERN :=, LIOP_SEL := #init, L_AUT := #init, L_REMOTE := #init, L_SIM :=, L_RESET := #reset, AUT_OP :=, MAN_OP :=, SIM_OP :=, FB_OPEN :=, FB_CLOSE :=, L_MON := #init, MON_T :=, MON_T_CLOSE :=, INSTANCE := 'AV-41.16', RESTART :=, VISIBILITY :=, OPdwCmd :=, QdwState =>, QwState =>, QCLOSING =>, QCLOSE =>, QOPENING =>, QOPEN =>, QCMD_OP => "AV-41.16", QMON =>, QMON_ERR =>, QMON_T =>, QMON_T_CLOSE =>, QMAN_AUT =>, QREMOTE =>, QSIM =>, QLOCK =>, QERR =>, QERR_EXT =>, QwAlarm =>)
   END_RUNG
   // the same network as SCL:
   #"AV-41.16"(LOCK := #"lock 3",   // "Valve"
               LIOP_SEL := #init,
               L_AUT := #init,
               L_REMOTE := #init,
               L_RESET := #reset,
               L_MON := #init,
               INSTANCE := 'AV-41.16',
               QCMD_OP => "AV-41.16");
END_REGION

REGION Network 20: AV-41.17 w ZSC
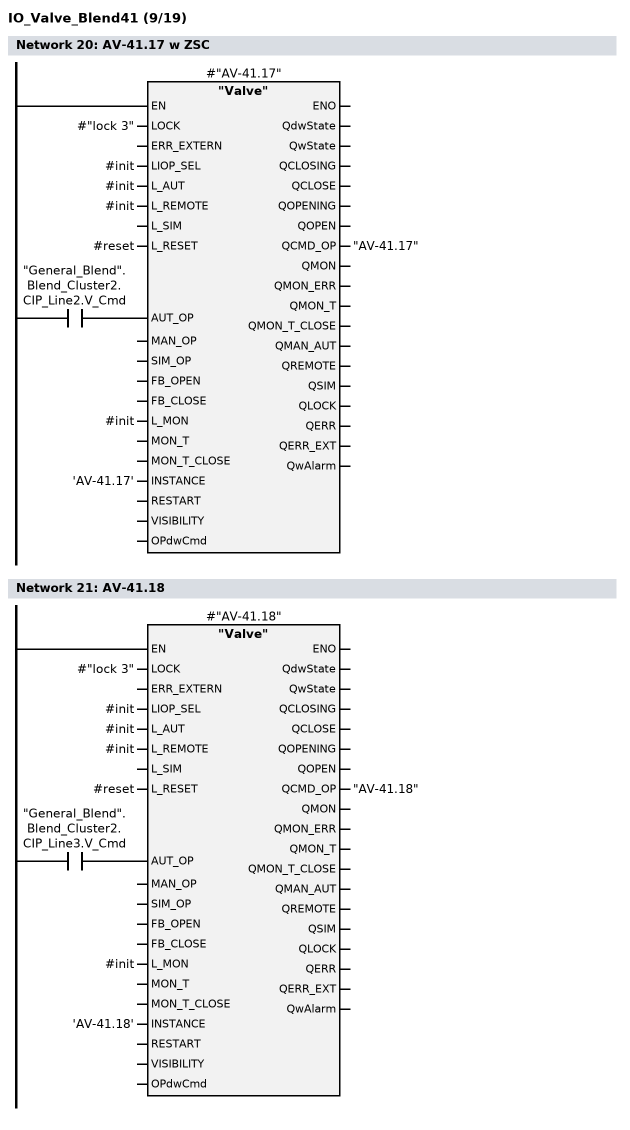
   RUNG wire#powerrail
      #"AV-41.17"(AUT_OP := wire#w1, LOCK := #"lock 3", ERR_EXTERN :=, LIOP_SEL := #init, L_AUT := #init, L_REMOTE := #init, L_SIM :=, L_RESET := #reset, MAN_OP :=, SIM_OP :=, FB_OPEN :=, FB_CLOSE :=, L_MON := #init, MON_T :=, MON_T_CLOSE :=, INSTANCE := 'AV-41.17', RESTART :=, VISIBILITY :=, OPdwCmd :=, QdwState =>, QwState =>, QCLOSING =>, QCLOSE =>, QOPENING =>, QOPEN =>, QCMD_OP => "AV-41.17", QMON =>, QMON_ERR =>, QMON_T =>, QMON_T_CLOSE =>, QMAN_AUT =>, QREMOTE =>, QSIM =>, QLOCK =>, QERR =>, QERR_EXT =>, QwAlarm =>)
   END_RUNG
   RUNG wire#powerrail
      Contact( "General_Blend".Blend_Cluster2.CIP_Line2.V_Cmd )
   END_RUNG wire#w1
   // the same network as SCL:
   #"AV-41.17"(LOCK := #"lock 3",   // "Valve"
               LIOP_SEL := #init,
               L_AUT := #init,
               L_REMOTE := #init,
               L_RESET := #reset,
               AUT_OP := "General_Blend".Blend_Cluster2.CIP_Line2.V_Cmd,
               L_MON := #init,
               INSTANCE := 'AV-41.17',
               QCMD_OP => "AV-41.17");
END_REGION

REGION Network 21: AV-41.18
   RUNG wire#powerrail
      #"AV-41.18"(AUT_OP := wire#w1, LOCK := #"lock 3", ERR_EXTERN :=, LIOP_SEL := #init, L_AUT := #init, L_REMOTE := #init, L_SIM :=, L_RESET := #reset, MAN_OP :=, SIM_OP :=, FB_OPEN :=, FB_CLOSE :=, L_MON := #init, MON_T :=, MON_T_CLOSE :=, INSTANCE := 'AV-41.18', RESTART :=, VISIBILITY :=, OPdwCmd :=, QdwState =>, QwState =>, QCLOSING =>, QCLOSE =>, QOPENING =>, QOPEN =>, QCMD_OP => "AV-41.18", QMON =>, QMON_ERR =>, QMON_T =>, QMON_T_CLOSE =>, QMAN_AUT =>, QREMOTE =>, QSIM =>, QLOCK =>, QERR =>, QERR_EXT =>, QwAlarm =>)
   END_RUNG
   RUNG wire#powerrail
      Contact( "General_Blend".Blend_Cluster2.CIP_Line3.V_Cmd )
   END_RUNG wire#w1
   // the same network as SCL:
   #"AV-41.18"(LOCK := #"lock 3",   // "Valve"
               LIOP_SEL := #init,
               L_AUT := #init,
               L_REMOTE := #init,
               L_RESET := #reset,
               AUT_OP := "General_Blend".Blend_Cluster2.CIP_Line3.V_Cmd,
               L_MON := #init,
               INSTANCE := 'AV-41.18',
               QCMD_OP => "AV-41.18");
END_REGION

REGION Network 22: AV-41.19
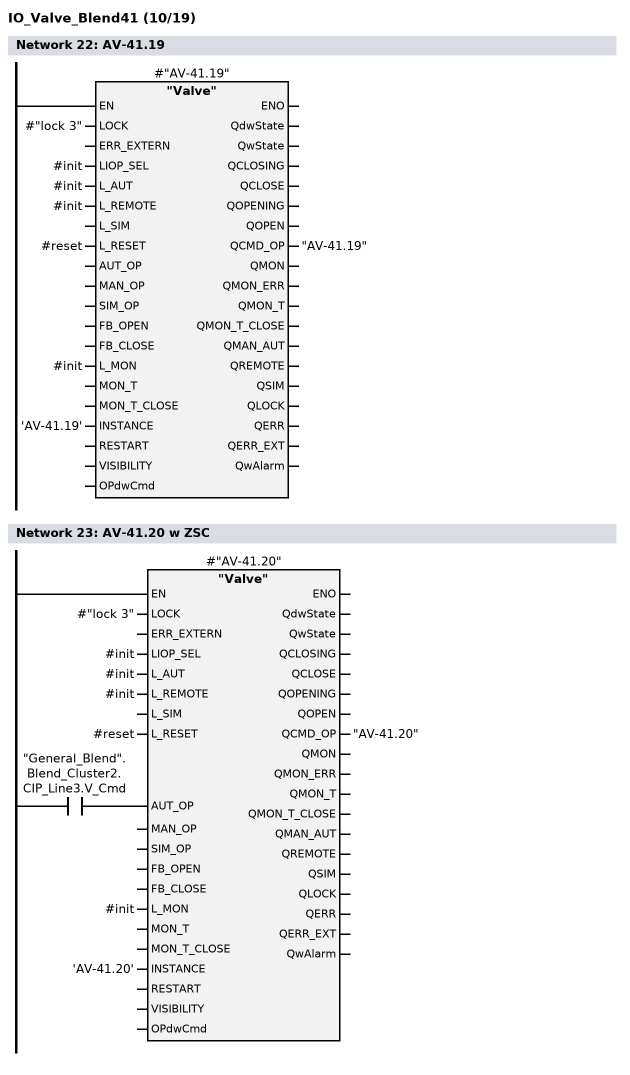
   RUNG wire#powerrail
      #"AV-41.19"(LOCK := #"lock 3", ERR_EXTERN :=, LIOP_SEL := #init, L_AUT := #init, L_REMOTE := #init, L_SIM :=, L_RESET := #reset, AUT_OP :=, MAN_OP :=, SIM_OP :=, FB_OPEN :=, FB_CLOSE :=, L_MON := #init, MON_T :=, MON_T_CLOSE :=, INSTANCE := 'AV-41.19', RESTART :=, VISIBILITY :=, OPdwCmd :=, QdwState =>, QwState =>, QCLOSING =>, QCLOSE =>, QOPENING =>, QOPEN =>, QCMD_OP => "AV-41.19", QMON =>, QMON_ERR =>, QMON_T =>, QMON_T_CLOSE =>, QMAN_AUT =>, QREMOTE =>, QSIM =>, QLOCK =>, QERR =>, QERR_EXT =>, QwAlarm =>)
   END_RUNG
   // the same network as SCL:
   #"AV-41.19"(LOCK := #"lock 3",   // "Valve"
               LIOP_SEL := #init,
               L_AUT := #init,
               L_REMOTE := #init,
               L_RESET := #reset,
               L_MON := #init,
               INSTANCE := 'AV-41.19',
               QCMD_OP => "AV-41.19");
END_REGION

REGION Network 23: AV-41.20 w ZSC
   RUNG wire#powerrail
      #"AV-41.20"(AUT_OP := wire#w1, LOCK := #"lock 3", ERR_EXTERN :=, LIOP_SEL := #init, L_AUT := #init, L_REMOTE := #init, L_SIM :=, L_RESET := #reset, MAN_OP :=, SIM_OP :=, FB_OPEN :=, FB_CLOSE :=, L_MON := #init, MON_T :=, MON_T_CLOSE :=, INSTANCE := 'AV-41.20', RESTART :=, VISIBILITY :=, OPdwCmd :=, QdwState =>, QwState =>, QCLOSING =>, QCLOSE =>, QOPENING =>, QOPEN =>, QCMD_OP => "AV-41.20", QMON =>, QMON_ERR =>, QMON_T =>, QMON_T_CLOSE =>, QMAN_AUT =>, QREMOTE =>, QSIM =>, QLOCK =>, QERR =>, QERR_EXT =>, QwAlarm =>)
   END_RUNG
   RUNG wire#powerrail
      Contact( "General_Blend".Blend_Cluster2.CIP_Line3.V_Cmd )
   END_RUNG wire#w1
   // the same network as SCL:
   #"AV-41.20"(LOCK := #"lock 3",   // "Valve"
               LIOP_SEL := #init,
               L_AUT := #init,
               L_REMOTE := #init,
               L_RESET := #reset,
               AUT_OP := "General_Blend".Blend_Cluster2.CIP_Line3.V_Cmd,
               L_MON := #init,
               INSTANCE := 'AV-41.20',
               QCMD_OP => "AV-41.20");
END_REGION

REGION Network 24: AV-41.21 w ZSC
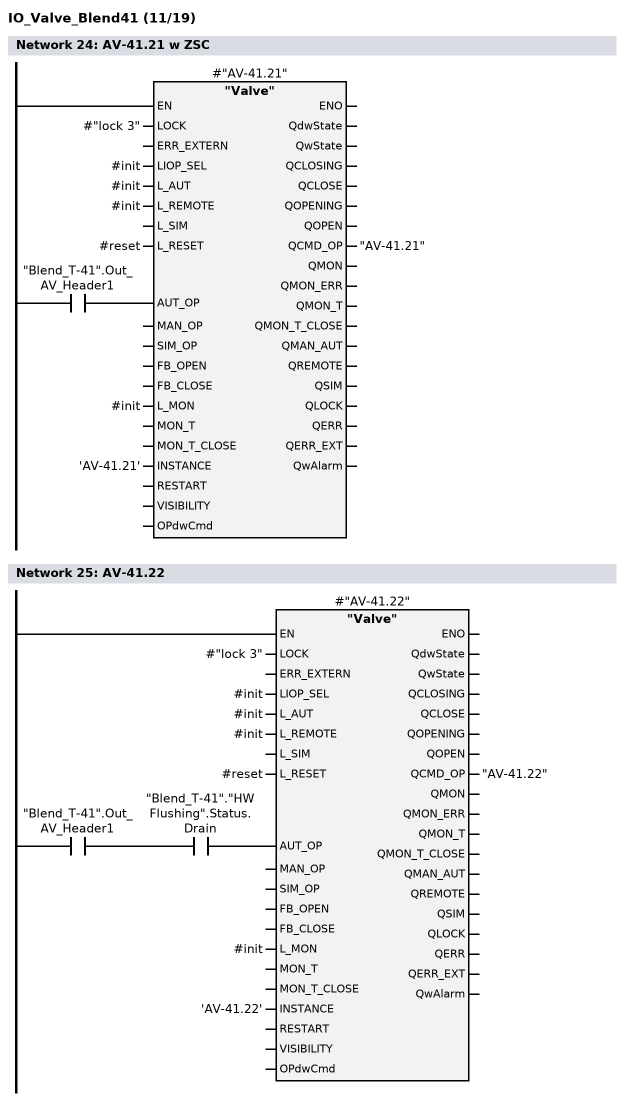
   RUNG wire#powerrail
      #"AV-41.21"(AUT_OP := wire#w1, LOCK := #"lock 3", ERR_EXTERN :=, LIOP_SEL := #init, L_AUT := #init, L_REMOTE := #init, L_SIM :=, L_RESET := #reset, MAN_OP :=, SIM_OP :=, FB_OPEN :=, FB_CLOSE :=, L_MON := #init, MON_T :=, MON_T_CLOSE :=, INSTANCE := 'AV-41.21', RESTART :=, VISIBILITY :=, OPdwCmd :=, QdwState =>, QwState =>, QCLOSING =>, QCLOSE =>, QOPENING =>, QOPEN =>, QCMD_OP => "AV-41.21", QMON =>, QMON_ERR =>, QMON_T =>, QMON_T_CLOSE =>, QMAN_AUT =>, QREMOTE =>, QSIM =>, QLOCK =>, QERR =>, QERR_EXT =>, QwAlarm =>)
   END_RUNG
   RUNG wire#powerrail
      Contact( "Blend_T-41".Out_AV_Header1 )
   END_RUNG wire#w1
   // the same network as SCL:
   #"AV-41.21"(LOCK := #"lock 3",   // "Valve"
               LIOP_SEL := #init,
               L_AUT := #init,
               L_REMOTE := #init,
               L_RESET := #reset,
               AUT_OP := "Blend_T-41".Out_AV_Header1,
               L_MON := #init,
               INSTANCE := 'AV-41.21',
               QCMD_OP => "AV-41.21");
END_REGION

REGION Network 25: AV-41.22
   RUNG wire#powerrail
      #"AV-41.22"(AUT_OP := wire#w1, LOCK := #"lock 3", ERR_EXTERN :=, LIOP_SEL := #init, L_AUT := #init, L_REMOTE := #init, L_SIM :=, L_RESET := #reset, MAN_OP :=, SIM_OP :=, FB_OPEN :=, FB_CLOSE :=, L_MON := #init, MON_T :=, MON_T_CLOSE :=, INSTANCE := 'AV-41.22', RESTART :=, VISIBILITY :=, OPdwCmd :=, QdwState =>, QwState =>, QCLOSING =>, QCLOSE =>, QOPENING =>, QOPEN =>, QCMD_OP => "AV-41.22", QMON =>, QMON_ERR =>, QMON_T =>, QMON_T_CLOSE =>, QMAN_AUT =>, QREMOTE =>, QSIM =>, QLOCK =>, QERR =>, QERR_EXT =>, QwAlarm =>)
   END_RUNG
   RUNG wire#powerrail
      Contact( "Blend_T-41".Out_AV_Header1 )
      Contact( "Blend_T-41"."HW Flushing".Status.Drain )
   END_RUNG wire#w1
   // the same network as SCL:
   #"AV-41.22"(LOCK := #"lock 3",   // "Valve"
               LIOP_SEL := #init,
               L_AUT := #init,
               L_REMOTE := #init,
               L_RESET := #reset,
               AUT_OP := "Blend_T-41".Out_AV_Header1 AND "Blend_T-41"."HW Flushing".Status.Drain,
               L_MON := #init,
               INSTANCE := 'AV-41.22',
               QCMD_OP => "AV-41.22");
END_REGION

REGION Network 26: AV-41.23 w ZSC
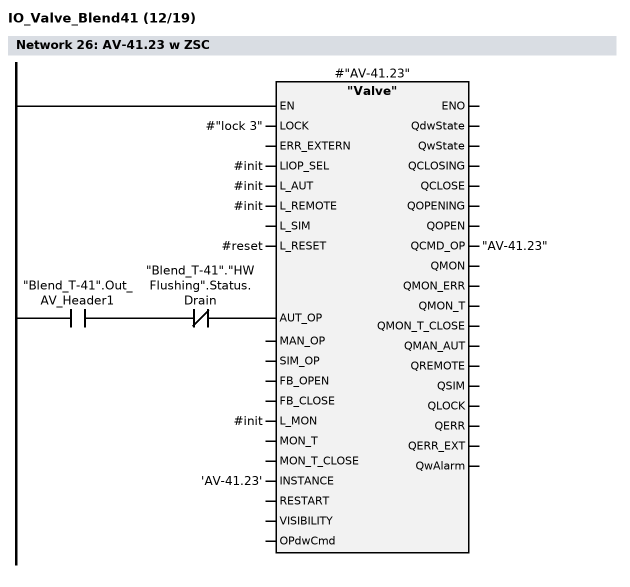
   RUNG wire#powerrail
      #"AV-41.23"(AUT_OP := wire#w1, LOCK := #"lock 3", ERR_EXTERN :=, LIOP_SEL := #init, L_AUT := #init, L_REMOTE := #init, L_SIM :=, L_RESET := #reset, MAN_OP :=, SIM_OP :=, FB_OPEN :=, FB_CLOSE :=, L_MON := #init, MON_T :=, MON_T_CLOSE :=, INSTANCE := 'AV-41.23', RESTART :=, VISIBILITY :=, OPdwCmd :=, QdwState =>, QwState =>, QCLOSING =>, QCLOSE =>, QOPENING =>, QOPEN =>, QCMD_OP => "AV-41.23", QMON =>, QMON_ERR =>, QMON_T =>, QMON_T_CLOSE =>, QMAN_AUT =>, QREMOTE =>, QSIM =>, QLOCK =>, QERR =>, QERR_EXT =>, QwAlarm =>)
   END_RUNG
   RUNG wire#powerrail
      Contact( "Blend_T-41".Out_AV_Header1 )
      I_Contact( "Blend_T-41"."HW Flushing".Status.Drain )
   END_RUNG wire#w1
   // the same network as SCL:
   #"AV-41.23"(LOCK := #"lock 3",   // "Valve"
               LIOP_SEL := #init,
               L_AUT := #init,
               L_REMOTE := #init,
               L_RESET := #reset,
               AUT_OP := "Blend_T-41".Out_AV_Header1 AND NOT "Blend_T-41"."HW Flushing".Status.Drain,
               L_MON := #init,
               INSTANCE := 'AV-41.23',
               QCMD_OP => "AV-41.23");
END_REGION

REGION Network 27: AV-41.24 w ZSC
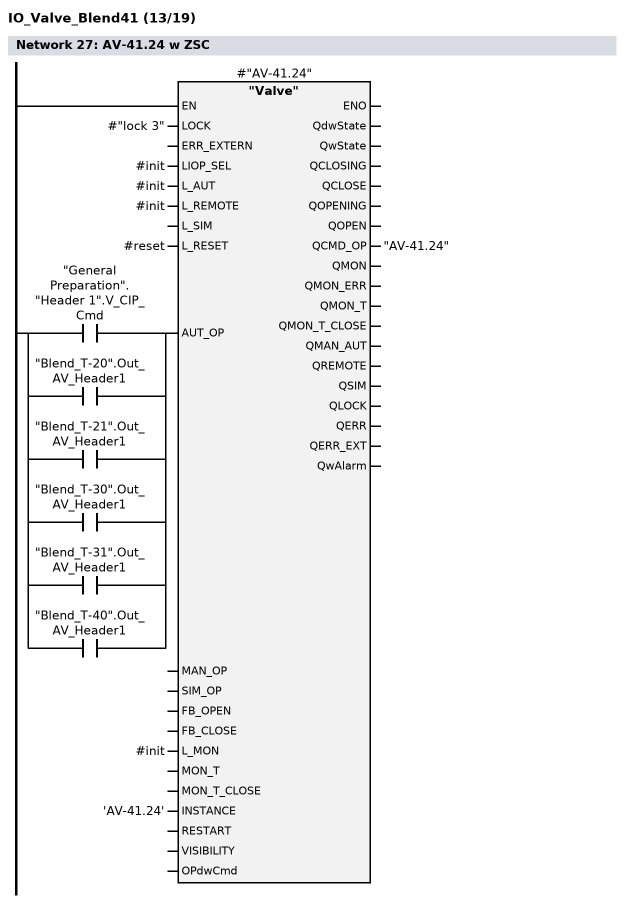
   RUNG wire#powerrail
      #"AV-41.24"(AUT_OP := wire#w1, LOCK := #"lock 3", ERR_EXTERN :=, LIOP_SEL := #init, L_AUT := #init, L_REMOTE := #init, L_SIM :=, L_RESET := #reset, MAN_OP :=, SIM_OP :=, FB_OPEN :=, FB_CLOSE :=, L_MON := #init, MON_T :=, MON_T_CLOSE :=, INSTANCE := 'AV-41.24', RESTART :=, VISIBILITY :=, OPdwCmd :=, QdwState =>, QwState =>, QCLOSING =>, QCLOSE =>, QOPENING =>, QOPEN =>, QCMD_OP => "AV-41.24", QMON =>, QMON_ERR =>, QMON_T =>, QMON_T_CLOSE =>, QMAN_AUT =>, QREMOTE =>, QSIM =>, QLOCK =>, QERR =>, QERR_EXT =>, QwAlarm =>)
   END_RUNG
   RUNG wire#powerrail
      Contact( "General Preparation"."Header 1".V_CIP_Cmd )
   END_RUNG wire#w1
   RUNG wire#powerrail
      Contact( "Blend_T-20".Out_AV_Header1 )
   END_RUNG wire#w1
   RUNG wire#powerrail
      Contact( "Blend_T-21".Out_AV_Header1 )
   END_RUNG wire#w1
   RUNG wire#powerrail
      Contact( "Blend_T-30".Out_AV_Header1 )
   END_RUNG wire#w1
   RUNG wire#powerrail
      Contact( "Blend_T-31".Out_AV_Header1 )
   END_RUNG wire#w1
   RUNG wire#powerrail
      Contact( "Blend_T-40".Out_AV_Header1 )
   END_RUNG wire#w1
   // the same network as SCL:
   #"AV-41.24"(LOCK := #"lock 3",   // "Valve"
               LIOP_SEL := #init,
               L_AUT := #init,
               L_REMOTE := #init,
               L_RESET := #reset,
               AUT_OP := "General Preparation"."Header 1".V_CIP_Cmd OR "Blend_T-20".Out_AV_Header1 OR "Blend_T-21".Out_AV_Header1 OR "Blend_T-30".Out_AV_Header1 OR "Blend_T-31".Out_AV_Header1 OR "Blend_T-40".Out_AV_Header1,
               L_MON := #init,
               INSTANCE := 'AV-41.24',
               QCMD_OP => "AV-41.24");
END_REGION

REGION Network 28: AV-41.25 w ZSC
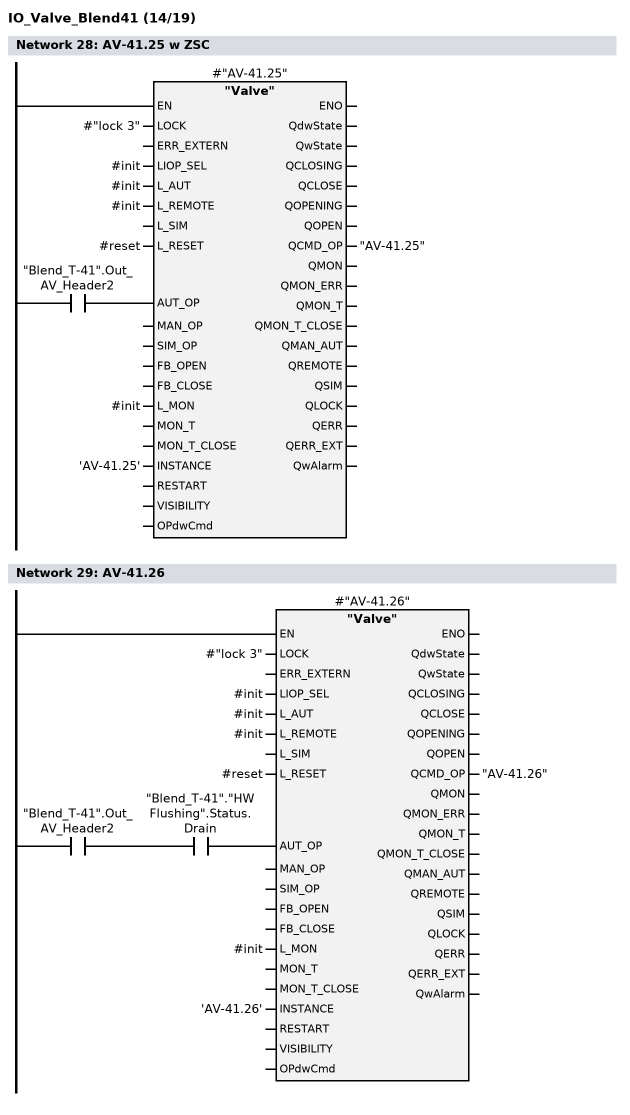
   RUNG wire#powerrail
      #"AV-41.25"(AUT_OP := wire#w1, LOCK := #"lock 3", ERR_EXTERN :=, LIOP_SEL := #init, L_AUT := #init, L_REMOTE := #init, L_SIM :=, L_RESET := #reset, MAN_OP :=, SIM_OP :=, FB_OPEN :=, FB_CLOSE :=, L_MON := #init, MON_T :=, MON_T_CLOSE :=, INSTANCE := 'AV-41.25', RESTART :=, VISIBILITY :=, OPdwCmd :=, QdwState =>, QwState =>, QCLOSING =>, QCLOSE =>, QOPENING =>, QOPEN =>, QCMD_OP => "AV-41.25", QMON =>, QMON_ERR =>, QMON_T =>, QMON_T_CLOSE =>, QMAN_AUT =>, QREMOTE =>, QSIM =>, QLOCK =>, QERR =>, QERR_EXT =>, QwAlarm =>)
   END_RUNG
   RUNG wire#powerrail
      Contact( "Blend_T-41".Out_AV_Header2 )
   END_RUNG wire#w1
   // the same network as SCL:
   #"AV-41.25"(LOCK := #"lock 3",   // "Valve"
               LIOP_SEL := #init,
               L_AUT := #init,
               L_REMOTE := #init,
               L_RESET := #reset,
               AUT_OP := "Blend_T-41".Out_AV_Header2,
               L_MON := #init,
               INSTANCE := 'AV-41.25',
               QCMD_OP => "AV-41.25");
END_REGION

REGION Network 29: AV-41.26
   RUNG wire#powerrail
      #"AV-41.26"(AUT_OP := wire#w1, LOCK := #"lock 3", ERR_EXTERN :=, LIOP_SEL := #init, L_AUT := #init, L_REMOTE := #init, L_SIM :=, L_RESET := #reset, MAN_OP :=, SIM_OP :=, FB_OPEN :=, FB_CLOSE :=, L_MON := #init, MON_T :=, MON_T_CLOSE :=, INSTANCE := 'AV-41.26', RESTART :=, VISIBILITY :=, OPdwCmd :=, QdwState =>, QwState =>, QCLOSING =>, QCLOSE =>, QOPENING =>, QOPEN =>, QCMD_OP => "AV-41.26", QMON =>, QMON_ERR =>, QMON_T =>, QMON_T_CLOSE =>, QMAN_AUT =>, QREMOTE =>, QSIM =>, QLOCK =>, QERR =>, QERR_EXT =>, QwAlarm =>)
   END_RUNG
   RUNG wire#powerrail
      Contact( "Blend_T-41".Out_AV_Header2 )
      Contact( "Blend_T-41"."HW Flushing".Status.Drain )
   END_RUNG wire#w1
   // the same network as SCL:
   #"AV-41.26"(LOCK := #"lock 3",   // "Valve"
               LIOP_SEL := #init,
               L_AUT := #init,
               L_REMOTE := #init,
               L_RESET := #reset,
               AUT_OP := "Blend_T-41".Out_AV_Header2 AND "Blend_T-41"."HW Flushing".Status.Drain,
               L_MON := #init,
               INSTANCE := 'AV-41.26',
               QCMD_OP => "AV-41.26");
END_REGION

REGION Network 30: AV-41.27 w ZSC
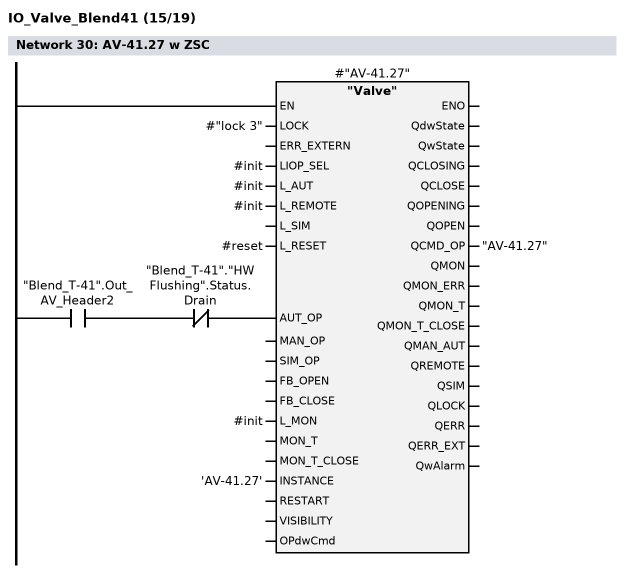
   RUNG wire#powerrail
      #"AV-41.27"(AUT_OP := wire#w1, LOCK := #"lock 3", ERR_EXTERN :=, LIOP_SEL := #init, L_AUT := #init, L_REMOTE := #init, L_SIM :=, L_RESET := #reset, MAN_OP :=, SIM_OP :=, FB_OPEN :=, FB_CLOSE :=, L_MON := #init, MON_T :=, MON_T_CLOSE :=, INSTANCE := 'AV-41.27', RESTART :=, VISIBILITY :=, OPdwCmd :=, QdwState =>, QwState =>, QCLOSING =>, QCLOSE =>, QOPENING =>, QOPEN =>, QCMD_OP => "AV-41.27", QMON =>, QMON_ERR =>, QMON_T =>, QMON_T_CLOSE =>, QMAN_AUT =>, QREMOTE =>, QSIM =>, QLOCK =>, QERR =>, QERR_EXT =>, QwAlarm =>)
   END_RUNG
   RUNG wire#powerrail
      Contact( "Blend_T-41".Out_AV_Header2 )
      I_Contact( "Blend_T-41"."HW Flushing".Status.Drain )
   END_RUNG wire#w1
   // the same network as SCL:
   #"AV-41.27"(LOCK := #"lock 3",   // "Valve"
               LIOP_SEL := #init,
               L_AUT := #init,
               L_REMOTE := #init,
               L_RESET := #reset,
               AUT_OP := "Blend_T-41".Out_AV_Header2 AND NOT "Blend_T-41"."HW Flushing".Status.Drain,
               L_MON := #init,
               INSTANCE := 'AV-41.27',
               QCMD_OP => "AV-41.27");
END_REGION

REGION Network 31: AV-41.28 w ZSC
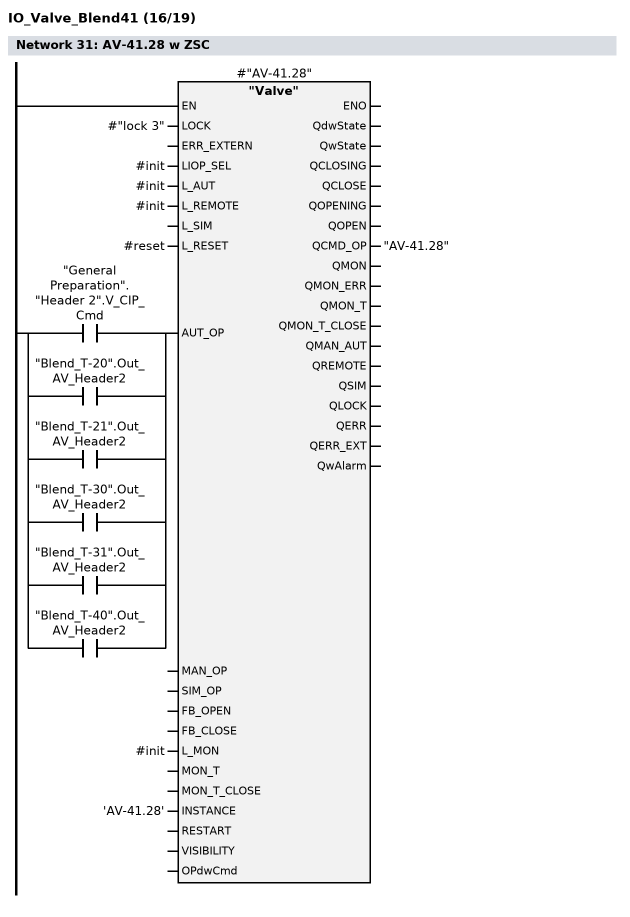
   RUNG wire#powerrail
      #"AV-41.28"(AUT_OP := wire#w1, LOCK := #"lock 3", ERR_EXTERN :=, LIOP_SEL := #init, L_AUT := #init, L_REMOTE := #init, L_SIM :=, L_RESET := #reset, MAN_OP :=, SIM_OP :=, FB_OPEN :=, FB_CLOSE :=, L_MON := #init, MON_T :=, MON_T_CLOSE :=, INSTANCE := 'AV-41.28', RESTART :=, VISIBILITY :=, OPdwCmd :=, QdwState =>, QwState =>, QCLOSING =>, QCLOSE =>, QOPENING =>, QOPEN =>, QCMD_OP => "AV-41.28", QMON =>, QMON_ERR =>, QMON_T =>, QMON_T_CLOSE =>, QMAN_AUT =>, QREMOTE =>, QSIM =>, QLOCK =>, QERR =>, QERR_EXT =>, QwAlarm =>)
   END_RUNG
   RUNG wire#powerrail
      Contact( "General Preparation"."Header 2".V_CIP_Cmd )
   END_RUNG wire#w1
   RUNG wire#powerrail
      Contact( "Blend_T-20".Out_AV_Header2 )
   END_RUNG wire#w1
   RUNG wire#powerrail
      Contact( "Blend_T-21".Out_AV_Header2 )
   END_RUNG wire#w1
   RUNG wire#powerrail
      Contact( "Blend_T-30".Out_AV_Header2 )
   END_RUNG wire#w1
   RUNG wire#powerrail
      Contact( "Blend_T-31".Out_AV_Header2 )
   END_RUNG wire#w1
   RUNG wire#powerrail
      Contact( "Blend_T-40".Out_AV_Header2 )
   END_RUNG wire#w1
   // the same network as SCL:
   #"AV-41.28"(LOCK := #"lock 3",   // "Valve"
               LIOP_SEL := #init,
               L_AUT := #init,
               L_REMOTE := #init,
               L_RESET := #reset,
               AUT_OP := "General Preparation"."Header 2".V_CIP_Cmd OR "Blend_T-20".Out_AV_Header2 OR "Blend_T-21".Out_AV_Header2 OR "Blend_T-30".Out_AV_Header2 OR "Blend_T-31".Out_AV_Header2 OR "Blend_T-40".Out_AV_Header2,
               L_MON := #init,
               INSTANCE := 'AV-41.28',
               QCMD_OP => "AV-41.28");
END_REGION

REGION Network 32: AV-41.29
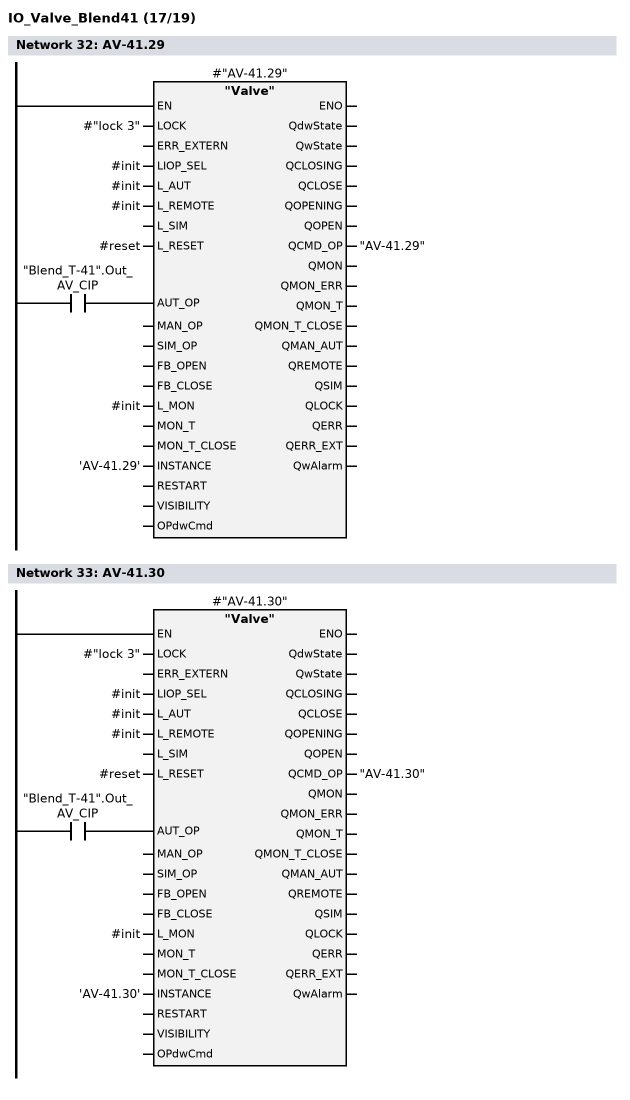
   RUNG wire#powerrail
      #"AV-41.29"(AUT_OP := wire#w1, LOCK := #"lock 3", ERR_EXTERN :=, LIOP_SEL := #init, L_AUT := #init, L_REMOTE := #init, L_SIM :=, L_RESET := #reset, MAN_OP :=, SIM_OP :=, FB_OPEN :=, FB_CLOSE :=, L_MON := #init, MON_T :=, MON_T_CLOSE :=, INSTANCE := 'AV-41.29', RESTART :=, VISIBILITY :=, OPdwCmd :=, QdwState =>, QwState =>, QCLOSING =>, QCLOSE =>, QOPENING =>, QOPEN =>, QCMD_OP => "AV-41.29", QMON =>, QMON_ERR =>, QMON_T =>, QMON_T_CLOSE =>, QMAN_AUT =>, QREMOTE =>, QSIM =>, QLOCK =>, QERR =>, QERR_EXT =>, QwAlarm =>)
   END_RUNG
   RUNG wire#powerrail
      Contact( "Blend_T-41".Out_AV_CIP )
   END_RUNG wire#w1
   // the same network as SCL:
   #"AV-41.29"(LOCK := #"lock 3",   // "Valve"
               LIOP_SEL := #init,
               L_AUT := #init,
               L_REMOTE := #init,
               L_RESET := #reset,
               AUT_OP := "Blend_T-41".Out_AV_CIP,
               L_MON := #init,
               INSTANCE := 'AV-41.29',
               QCMD_OP => "AV-41.29");
END_REGION

REGION Network 33: AV-41.30
   RUNG wire#powerrail
      #"AV-41.30"(AUT_OP := wire#w1, LOCK := #"lock 3", ERR_EXTERN :=, LIOP_SEL := #init, L_AUT := #init, L_REMOTE := #init, L_SIM :=, L_RESET := #reset, MAN_OP :=, SIM_OP :=, FB_OPEN :=, FB_CLOSE :=, L_MON := #init, MON_T :=, MON_T_CLOSE :=, INSTANCE := 'AV-41.30', RESTART :=, VISIBILITY :=, OPdwCmd :=, QdwState =>, QwState =>, QCLOSING =>, QCLOSE =>, QOPENING =>, QOPEN =>, QCMD_OP => "AV-41.30", QMON =>, QMON_ERR =>, QMON_T =>, QMON_T_CLOSE =>, QMAN_AUT =>, QREMOTE =>, QSIM =>, QLOCK =>, QERR =>, QERR_EXT =>, QwAlarm =>)
   END_RUNG
   RUNG wire#powerrail
      Contact( "Blend_T-41".Out_AV_CIP )
   END_RUNG wire#w1
   // the same network as SCL:
   #"AV-41.30"(LOCK := #"lock 3",   // "Valve"
               LIOP_SEL := #init,
               L_AUT := #init,
               L_REMOTE := #init,
               L_RESET := #reset,
               AUT_OP := "Blend_T-41".Out_AV_CIP,
               L_MON := #init,
               INSTANCE := 'AV-41.30',
               QCMD_OP => "AV-41.30");
END_REGION

REGION Network 34: AV-41.31 w ZSC
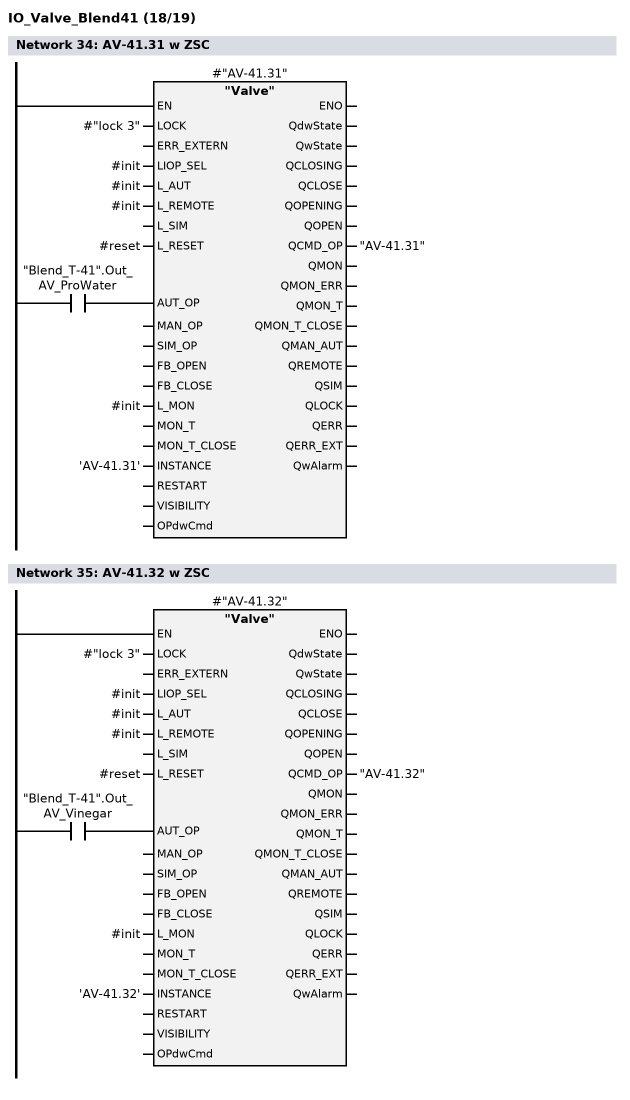
   RUNG wire#powerrail
      #"AV-41.31"(AUT_OP := wire#w1, LOCK := #"lock 3", ERR_EXTERN :=, LIOP_SEL := #init, L_AUT := #init, L_REMOTE := #init, L_SIM :=, L_RESET := #reset, MAN_OP :=, SIM_OP :=, FB_OPEN :=, FB_CLOSE :=, L_MON := #init, MON_T :=, MON_T_CLOSE :=, INSTANCE := 'AV-41.31', RESTART :=, VISIBILITY :=, OPdwCmd :=, QdwState =>, QwState =>, QCLOSING =>, QCLOSE =>, QOPENING =>, QOPEN =>, QCMD_OP => "AV-41.31", QMON =>, QMON_ERR =>, QMON_T =>, QMON_T_CLOSE =>, QMAN_AUT =>, QREMOTE =>, QSIM =>, QLOCK =>, QERR =>, QERR_EXT =>, QwAlarm =>)
   END_RUNG
   RUNG wire#powerrail
      Contact( "Blend_T-41".Out_AV_ProWater )
   END_RUNG wire#w1
   // the same network as SCL:
   #"AV-41.31"(LOCK := #"lock 3",   // "Valve"
               LIOP_SEL := #init,
               L_AUT := #init,
               L_REMOTE := #init,
               L_RESET := #reset,
               AUT_OP := "Blend_T-41".Out_AV_ProWater,
               L_MON := #init,
               INSTANCE := 'AV-41.31',
               QCMD_OP => "AV-41.31");
END_REGION

REGION Network 35: AV-41.32 w ZSC
   RUNG wire#powerrail
      #"AV-41.32"(AUT_OP := wire#w1, LOCK := #"lock 3", ERR_EXTERN :=, LIOP_SEL := #init, L_AUT := #init, L_REMOTE := #init, L_SIM :=, L_RESET := #reset, MAN_OP :=, SIM_OP :=, FB_OPEN :=, FB_CLOSE :=, L_MON := #init, MON_T :=, MON_T_CLOSE :=, INSTANCE := 'AV-41.32', RESTART :=, VISIBILITY :=, OPdwCmd :=, QdwState =>, QwState =>, QCLOSING =>, QCLOSE =>, QOPENING =>, QOPEN =>, QCMD_OP => "AV-41.32", QMON =>, QMON_ERR =>, QMON_T =>, QMON_T_CLOSE =>, QMAN_AUT =>, QREMOTE =>, QSIM =>, QLOCK =>, QERR =>, QERR_EXT =>, QwAlarm =>)
   END_RUNG
   RUNG wire#powerrail
      Contact( "Blend_T-41".Out_AV_Vinegar )
   END_RUNG wire#w1
   // the same network as SCL:
   #"AV-41.32"(LOCK := #"lock 3",   // "Valve"
               LIOP_SEL := #init,
               L_AUT := #init,
               L_REMOTE := #init,
               L_RESET := #reset,
               AUT_OP := "Blend_T-41".Out_AV_Vinegar,
               L_MON := #init,
               INSTANCE := 'AV-41.32',
               QCMD_OP => "AV-41.32");
END_REGION

REGION Network 36: AV-41.33 w ZSC
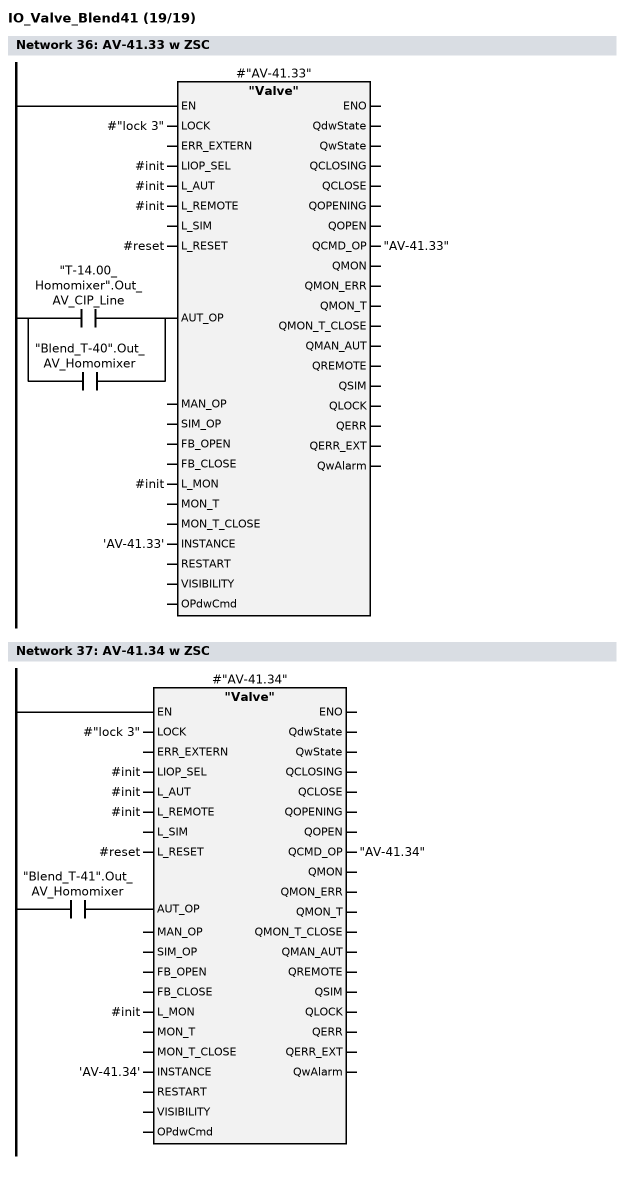
   RUNG wire#powerrail
      #"AV-41.33"(AUT_OP := wire#w1, LOCK := #"lock 3", ERR_EXTERN :=, LIOP_SEL := #init, L_AUT := #init, L_REMOTE := #init, L_SIM :=, L_RESET := #reset, MAN_OP :=, SIM_OP :=, FB_OPEN :=, FB_CLOSE :=, L_MON := #init, MON_T :=, MON_T_CLOSE :=, INSTANCE := 'AV-41.33', RESTART :=, VISIBILITY :=, OPdwCmd :=, QdwState =>, QwState =>, QCLOSING =>, QCLOSE =>, QOPENING =>, QOPEN =>, QCMD_OP => "AV-41.33", QMON =>, QMON_ERR =>, QMON_T =>, QMON_T_CLOSE =>, QMAN_AUT =>, QREMOTE =>, QSIM =>, QLOCK =>, QERR =>, QERR_EXT =>, QwAlarm =>)
   END_RUNG
   RUNG wire#powerrail
      Contact( "T-14.00_Homomixer".Out_AV_CIP_Line )
   END_RUNG wire#w1
   RUNG wire#powerrail
      Contact( "Blend_T-40".Out_AV_Homomixer )
   END_RUNG wire#w1
   // the same network as SCL:
   #"AV-41.33"(LOCK := #"lock 3",   // "Valve"
               LIOP_SEL := #init,
               L_AUT := #init,
               L_REMOTE := #init,
               L_RESET := #reset,
               AUT_OP := "T-14.00_Homomixer".Out_AV_CIP_Line OR "Blend_T-40".Out_AV_Homomixer,
               L_MON := #init,
               INSTANCE := 'AV-41.33',
               QCMD_OP => "AV-41.33");
END_REGION

REGION Network 37: AV-41.34 w ZSC
   RUNG wire#powerrail
      #"AV-41.34"(AUT_OP := wire#w1, LOCK := #"lock 3", ERR_EXTERN :=, LIOP_SEL := #init, L_AUT := #init, L_REMOTE := #init, L_SIM :=, L_RESET := #reset, MAN_OP :=, SIM_OP :=, FB_OPEN :=, FB_CLOSE :=, L_MON := #init, MON_T :=, MON_T_CLOSE :=, INSTANCE := 'AV-41.34', RESTART :=, VISIBILITY :=, OPdwCmd :=, QdwState =>, QwState =>, QCLOSING =>, QCLOSE =>, QOPENING =>, QOPEN =>, QCMD_OP => "AV-41.34", QMON =>, QMON_ERR =>, QMON_T =>, QMON_T_CLOSE =>, QMAN_AUT =>, QREMOTE =>, QSIM =>, QLOCK =>, QERR =>, QERR_EXT =>, QwAlarm =>)
   END_RUNG
   RUNG wire#powerrail
      Contact( "Blend_T-41".Out_AV_Homomixer )
   END_RUNG wire#w1
   // the same network as SCL:
   #"AV-41.34"(LOCK := #"lock 3",   // "Valve"
               LIOP_SEL := #init,
               L_AUT := #init,
               L_REMOTE := #init,
               L_RESET := #reset,
               AUT_OP := "Blend_T-41".Out_AV_Homomixer,
               L_MON := #init,
               INSTANCE := 'AV-41.34',
               QCMD_OP => "AV-41.34");
END_REGION
END_FUNCTION_BLOCK

FUNCTION "IO Storage" : Void   // FC4, LAD
{ S7_Optimized_Access := 'TRUE' }
VERSION : 0.1
// stored: AutoNumber true, IsIECCheckEnabled false, SetENOAutomatically false, UDAEnableTagReadback false
   VAR_TEMP   // added for the SCL form of the ladder/FBD networks
      _w1 : Bool;
      _w2 : Bool;
      _w3 : Bool;
      _w4 : Bool;
   END_VAR
BEGIN

REGION Network 1: Analog IO
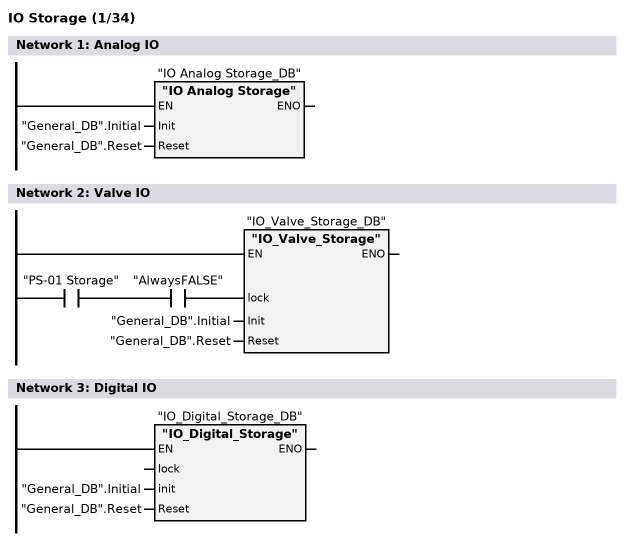
   RUNG wire#powerrail
      "IO Analog Storage_DB"(Init := "General_DB".Initial, Reset := "General_DB".Reset)
   END_RUNG
   // the same network as SCL:
   "IO Analog Storage_DB"(Init := "General_DB".Initial, Reset := "General_DB".Reset);   // "IO Analog Storage"
END_REGION

REGION Network 2: Valve IO
   RUNG wire#powerrail
      "IO_Valve_Storage_DB"(lock := wire#w1, Init := "General_DB".Initial, Reset := "General_DB".Reset)
   END_RUNG
   RUNG wire#powerrail
      Contact( "PS-01 Storage" )
      Contact( "AlwaysFALSE" )
   END_RUNG wire#w1
   // the same network as SCL:
   "IO_Valve_Storage_DB"(lock := "PS-01 Storage" AND "AlwaysFALSE",   // "IO_Valve_Storage"
                         Init := "General_DB".Initial,
                         Reset := "General_DB".Reset);
END_REGION

REGION Network 3: Digital IO
   RUNG wire#powerrail
      "IO_Digital_Storage_DB"(lock :=, init := "General_DB".Initial, Reset := "General_DB".Reset)
   END_RUNG
   // the same network as SCL:
   "IO_Digital_Storage_DB"(init := "General_DB".Initial, Reset := "General_DB".Reset);   // "IO_Digital_Storage"
END_REGION

REGION Network 4 (SCL): Bypass CIP Signal
   IF "General_DB"."Bypass CIP Signal Storage" = TRUE THEN
       // T-29 JBT
       //"T-29.00".CIP_Req_OK := TRUE;
       //"T-29.00".CIP_ON_Progress := TRUE;
       //"T-29.00".CIP_Supply_ON := TRUE;
       //"T-29.00".CIP_Complete := FALSE;
       // T-23
       "T-23.00".CIP_Req_OK := TRUE;
       "T-23.00".CIP_ON_Progress := TRUE;
       "T-23.00".CIP_Supply_ON := TRUE;
       "T-23.00".CIP_Complete := FALSE;
       // T-24
       "T-24.00".CIP_Req_OK := TRUE;
       "T-24.00".CIP_ON_Progress := TRUE;
       "T-24.00".CIP_Supply_ON := TRUE;
       "T-24.00".CIP_Complete := FALSE;
       // T-39 JBT
       //"T-39.00".CIP_Req_OK := TRUE;
       //"T-39.00".CIP_ON_Progress := TRUE;
       //"T-39.00".CIP_Supply_ON := TRUE;
       //"T-39.00".CIP_Complete := FALSE;
       // T-33
       "T-33.00".CIP_Req_OK := TRUE;
       "T-33.00".CIP_ON_Progress := TRUE;
       "T-33.00".CIP_Supply_ON := TRUE;
       "T-33.00".CIP_Complete := FALSE;
       // T-34
       "T-34.00".CIP_Req_OK := TRUE;
       "T-34.00".CIP_ON_Progress := TRUE;
       "T-34.00".CIP_Supply_ON := TRUE;
       "T-34.00".CIP_Complete := FALSE;
       // T-35
       "T-35.00".CIP_Req_OK := TRUE;
       "T-35.00".CIP_ON_Progress := TRUE;
       "T-35.00".CIP_Supply_ON := TRUE;
       "T-35.00".CIP_Complete := FALSE;
       // T-79
       "T-79.00".CIP_Req_OK:= TRUE;
       "T-79.00".CIP_ON_Progress:= TRUE;
       "T-79.00".CIP_Supply_ON:= TRUE;
       "T-79.00".CIP_Complete:= FALSE;
       // T-81
       "T-81.00".CIP_Req_OK := TRUE;
       "T-81.00".CIP_ON_Progress := TRUE;
       "T-81.00".CIP_Supply_ON := TRUE;
       "T-81.00".CIP_Complete := FALSE;
       // T-84
       "T-84.00".CIP_Req_OK := TRUE;
       "T-84.00".CIP_ON_Progress := TRUE;
       "T-84.00".CIP_Supply_ON := TRUE;
       "T-84.00".CIP_Complete := FALSE;
       // T-85
       "T-85.00".CIP_Req_OK := TRUE;
       "T-85.00".CIP_ON_Progress := TRUE;
       "T-85.00".CIP_Supply_ON := TRUE;
       "T-85.00".CIP_Complete := FALSE;
   ELSE
       // T-29 JBT
       //"T-29.00".CIP_Req_OK := "CIP_to_Mix".CIP_RequestOK."Storage THE 4".THE4_LineProduct_CIP_RequestOK;
       //"T-29.00".CIP_ON_Progress := "CIP_to_Mix".CIP_InProgress."Storage THE 4".THE4_LineProduct_CIP_InProgress;
       //"T-29.00".CIP_Supply_ON := "CIP_to_Mix".CIP_Supply_On."Storage THE 4".THE4_LineProduct_CIP_Supply_ON;
       //"T-29.00".CIP_Complete := "CIP_to_Mix".CIP_Complete."Storage THE 4".THE4_LineProduct_CIP_Complete;
       // T-23
       "T-23.00".CIP_Req_OK := "CIP_to_Mix".CIP_RequestOK."Storage THE 4"."T-23.00_CIP_RequestOK";
       "T-23.00".CIP_ON_Progress := "CIP_to_Mix".CIP_InProgress."Storage THE 4"."T-23.00_CIP_InProgress";
       "T-23.00".CIP_Supply_ON := "CIP_to_Mix".CIP_Supply_On."Storage THE 4"."T-23.00_CIP_Supply_ON";
       "T-23.00".CIP_Complete := "CIP_to_Mix".CIP_Complete."Storage THE 4"."T-23.00_CIP_Complete";
       // T-24
       "T-24.00".CIP_Req_OK := "CIP_to_Mix".CIP_RequestOK."Storage THE 4"."T-24.00_CIP_RequestOK";
       "T-24.00".CIP_ON_Progress := "CIP_to_Mix".CIP_InProgress."Storage THE 4"."T-24.00_CIP_InProgress";
       "T-24.00".CIP_Supply_ON := "CIP_to_Mix".CIP_Supply_On."Storage THE 4"."T-24.00_CIP_Supply_ON";
       "T-24.00".CIP_Complete := "CIP_to_Mix".CIP_Complete."Storage THE 4"."T-24.00_CIP_Complete";
       // T-39 JBT
       //"T-39.00".CIP_Req_OK := "CIP_to_Mix".CIP_RequestOK."Storage THE 5".THE5_LineProduct_CIP_RequestOK;
       //"T-39.00".CIP_ON_Progress := "CIP_to_Mix".CIP_InProgress."Storage THE 5".THE5_LineProduct_CIP_InProgress;
       //"T-39.00".CIP_Supply_ON := "CIP_to_Mix".CIP_Supply_On."Storage THE 5".THE5_LineProduct_CIP_Supply_ON;
       //"T-39.00".CIP_Complete := "CIP_to_Mix".CIP_Complete."Storage THE 5".THE5_LineProduct_CIP_Complete;
       // T-33
       "T-33.00".CIP_Req_OK := "CIP_to_Mix".CIP_RequestOK."Storage THE 5"."T-33.00_CIP_Tank_RequestOK" OR "CIP_to_Mix".CIP_RequestOK."Storage THE 5"."T33&T34_CIP_Line_RequestOK";
       "T-33.00".CIP_ON_Progress := "CIP_to_Mix".CIP_InProgress."Storage THE 5"."T-33.00_CIP_Tank_InProgress" OR "CIP_to_Mix".CIP_InProgress."Storage THE 5"."T33&T34_CIP_Line_InProgress";
       "T-33.00".CIP_Supply_ON := "CIP_to_Mix".CIP_Supply_On."Storage THE 5"."T-33.00_CIP_Tank_Supply_ON" OR "CIP_to_Mix".CIP_Supply_On."Storage THE 5"."T33&T34_CIP_Line_Supply_ON";
       "T-33.00".CIP_Complete := "CIP_to_Mix".CIP_Complete."Storage THE 5"."T-33.00_CIP_Tank_Complete" OR "CIP_to_Mix".CIP_Complete."Storage THE 5"."T33&T34_CIP_Line_Complete";
       // T-34
       "T-34.00".CIP_Req_OK := "CIP_to_Mix".CIP_RequestOK."Storage THE 5"."T-34.00_CIP_Tank_RequestOK" OR "CIP_to_Mix".CIP_RequestOK."Storage THE 5"."T33&T34_CIP_Line_RequestOK";
       "T-34.00".CIP_ON_Progress := "CIP_to_Mix".CIP_InProgress."Storage THE 5"."T-34.00_CIP_Tank_InProgress" OR "CIP_to_Mix".CIP_InProgress."Storage THE 5"."T33&T34_CIP_Line_InProgress";
       "T-34.00".CIP_Supply_ON := "CIP_to_Mix".CIP_Supply_On."Storage THE 5"."T-34.00_CIP_Tank_Supply_ON" OR "CIP_to_Mix".CIP_Supply_On."Storage THE 5"."T33&T34_CIP_Line_Supply_ON";
       "T-34.00".CIP_Complete := "CIP_to_Mix".CIP_Complete."Storage THE 5"."T-34.00_CIP_Tank_Complete" OR "CIP_to_Mix".CIP_Complete."Storage THE 5"."T33&T34_CIP_Line_Complete";
       // T-35
       "T-35.00".CIP_Req_OK := "CIP_to_Mix".CIP_RequestOK."Storage THE 5"."T-35.00_CIP_Tank_RequestOK";
       "T-35.00".CIP_ON_Progress := "CIP_to_Mix".CIP_InProgress."Storage THE 5"."T-35.00_CIP_Tank_InProgress";
       "T-35.00".CIP_Supply_ON := "CIP_to_Mix".CIP_Supply_On."Storage THE 5"."T-35.00_CIP_Tank_Supply_ON";
       "T-35.00".CIP_Complete := "CIP_to_Mix".CIP_Complete."Storage THE 5"."T-35.00_CIP_Tank_Complete";
       // T-79
       "T-79.00".CIP_Req_OK:= "CIP_to_Mix".CIP_RequestOK."T-79.00_CIP_RequestOK";
       "T-79.00".CIP_ON_Progress:= "CIP_to_Mix".CIP_InProgress."T-79.00_CIP_InProgress";
       "T-79.00".CIP_Supply_ON:= "CIP_to_Mix".CIP_Supply_On."T-79.00_CIP_Supply_ON";
       "T-79.00".CIP_Complete := "CIP_to_Mix".CIP_Complete."T-79.00_CIP_Complete";
       // T-81
       "T-81.00".CIP_Req_OK := "CIP_to_Mix".CIP_RequestOK."T-81.00_CIP_RequestOK";
       "T-81.00".CIP_ON_Progress := "CIP_to_Mix".CIP_InProgress."T-81.00_CIP_InProgress";
       "T-81.00".CIP_Supply_ON := "CIP_to_Mix".CIP_Supply_On."T-81.00_CIP_Supply_ON";
       "T-81.00".CIP_Complete := "CIP_to_Mix".CIP_Complete."T-81.00_CIP_Complete";
       // T-84
       "T-84.00".CIP_Req_OK := "CIP_to_Mix".CIP_RequestOK."T-84.00_CIP_RequestOK";
       "T-84.00".CIP_ON_Progress := "CIP_to_Mix".CIP_InProgress."T-84.00_CIP_InProgress";
       "T-84.00".CIP_Supply_ON := "CIP_to_Mix".CIP_Supply_On."T-84.00_CIP_Supply_ON";
       "T-84.00".CIP_Complete := "CIP_to_Mix".CIP_Complete."T-84.00_CIP_Complete";
       // T-85
       "T-85.00".CIP_Req_OK := "CIP_to_Mix".CIP_RequestOK."T-85.00_CIP_RequestOK";
       "T-85.00".CIP_ON_Progress := "CIP_to_Mix".CIP_InProgress."T-85.00_CIP_InProgress";
       "T-85.00".CIP_Supply_ON := "CIP_to_Mix".CIP_Supply_On."T-85.00_CIP_Supply_ON";
       "T-85.00".CIP_Complete := "CIP_to_Mix".CIP_Complete."T-85.00_CIP_Complete";
   END_IF;
END_REGION

REGION Network 6: T-29.00 ST-03 -> Tank Storage By JBT
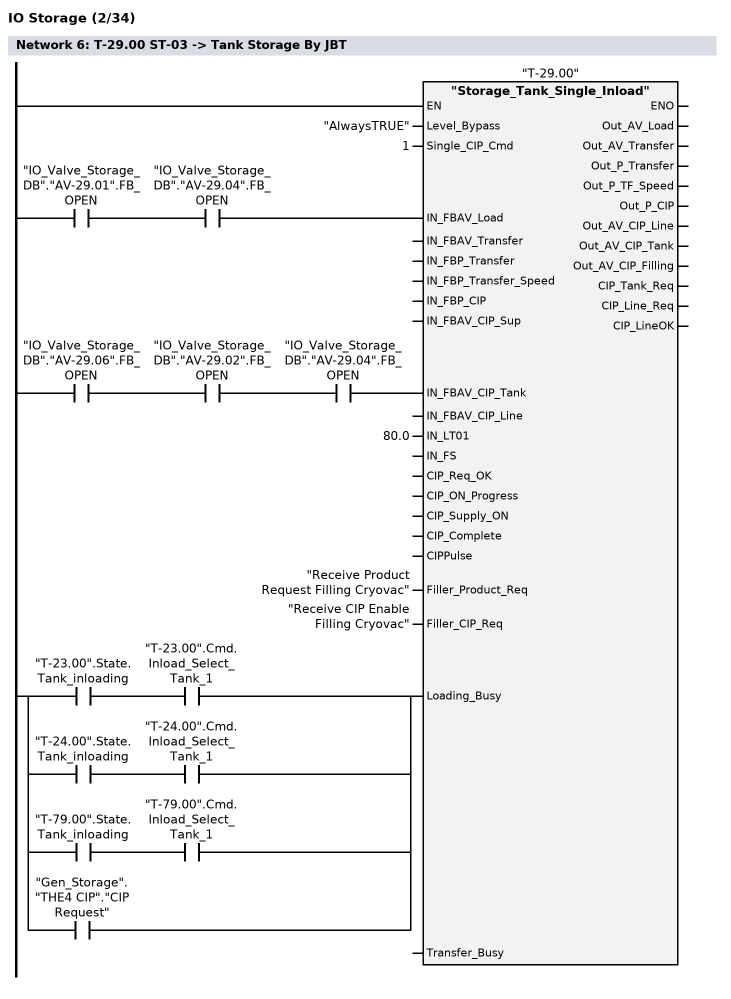
   RUNG wire#powerrail
      "T-29.00"(IN_FBAV_Load := wire#w1, IN_FBAV_CIP_Tank := wire#w2, Loading_Busy := wire#w3, Level_Bypass := "AlwaysTRUE", Single_CIP_Cmd := 1, IN_FBAV_Transfer :=, IN_FBP_Transfer :=, IN_FBP_Transfer_Speed :=, IN_FBP_CIP :=, IN_FBAV_CIP_Sup :=, IN_FBAV_CIP_Line :=, IN_LT01 := 80.0, IN_FS :=, CIP_Req_OK :=, CIP_ON_Progress :=, CIP_Supply_ON :=, CIP_Complete :=, CIPPulse :=, Filler_Product_Req := "Receive Product Request Filling Cryovac", Filler_CIP_Req := "Receive CIP Enable Filling Cryovac", Transfer_Busy :=, Out_AV_Load =>, Out_AV_Transfer =>, Out_P_Transfer =>, Out_P_TF_Speed =>, Out_P_CIP =>, Out_AV_CIP_Line =>, Out_AV_CIP_Tank =>, Out_AV_CIP_Filling =>, CIP_Tank_Req =>, CIP_Line_Req =>, CIP_LineOK =>)
   END_RUNG
   RUNG wire#powerrail
      Contact( "IO_Valve_Storage_DB"."AV-29.01".FB_OPEN )
      Contact( "IO_Valve_Storage_DB"."AV-29.04".FB_OPEN )
   END_RUNG wire#w1
   RUNG wire#powerrail
      Contact( "IO_Valve_Storage_DB"."AV-29.06".FB_OPEN )
      Contact( "IO_Valve_Storage_DB"."AV-29.02".FB_OPEN )
      Contact( "IO_Valve_Storage_DB"."AV-29.04".FB_OPEN )
   END_RUNG wire#w2
   RUNG wire#powerrail
      Contact( "T-23.00".State.Tank_inloading )
      Contact( "T-23.00".Cmd.Inload_Select_Tank_1 )
   END_RUNG wire#w3
   RUNG wire#powerrail
      Contact( "T-24.00".State.Tank_inloading )
      Contact( "T-24.00".Cmd.Inload_Select_Tank_1 )
   END_RUNG wire#w3
   RUNG wire#powerrail
      Contact( "T-79.00".State.Tank_inloading )
      Contact( "T-79.00".Cmd.Inload_Select_Tank_1 )
   END_RUNG wire#w3
   RUNG wire#powerrail
      Contact( "Gen_Storage"."THE4 CIP"."CIP Request" )
   END_RUNG wire#w3
   // the same network as SCL:
   "T-29.00"(Level_Bypass := "AlwaysTRUE",   // "Storage_Tank_Single_Inload"
             Single_CIP_Cmd := 1,
             IN_FBAV_Load := "IO_Valve_Storage_DB"."AV-29.01".FB_OPEN AND "IO_Valve_Storage_DB"."AV-29.04".FB_OPEN,
             IN_FBAV_CIP_Tank := "IO_Valve_Storage_DB"."AV-29.06".FB_OPEN AND "IO_Valve_Storage_DB"."AV-29.02".FB_OPEN AND "IO_Valve_Storage_DB"."AV-29.04".FB_OPEN,
             IN_LT01 := 80.0,
             Filler_Product_Req := "Receive Product Request Filling Cryovac",
             Filler_CIP_Req := "Receive CIP Enable Filling Cryovac",
             Loading_Busy := ("T-23.00".State.Tank_inloading AND "T-23.00".Cmd.Inload_Select_Tank_1) OR ("T-24.00".State.Tank_inloading AND "T-24.00".Cmd.Inload_Select_Tank_1) OR ("T-79.00".State.Tank_inloading AND "T-79.00".Cmd.Inload_Select_Tank_1) OR "Gen_Storage"."THE4 CIP"."CIP Request");
END_REGION

REGION Network 7: T-29 Valve
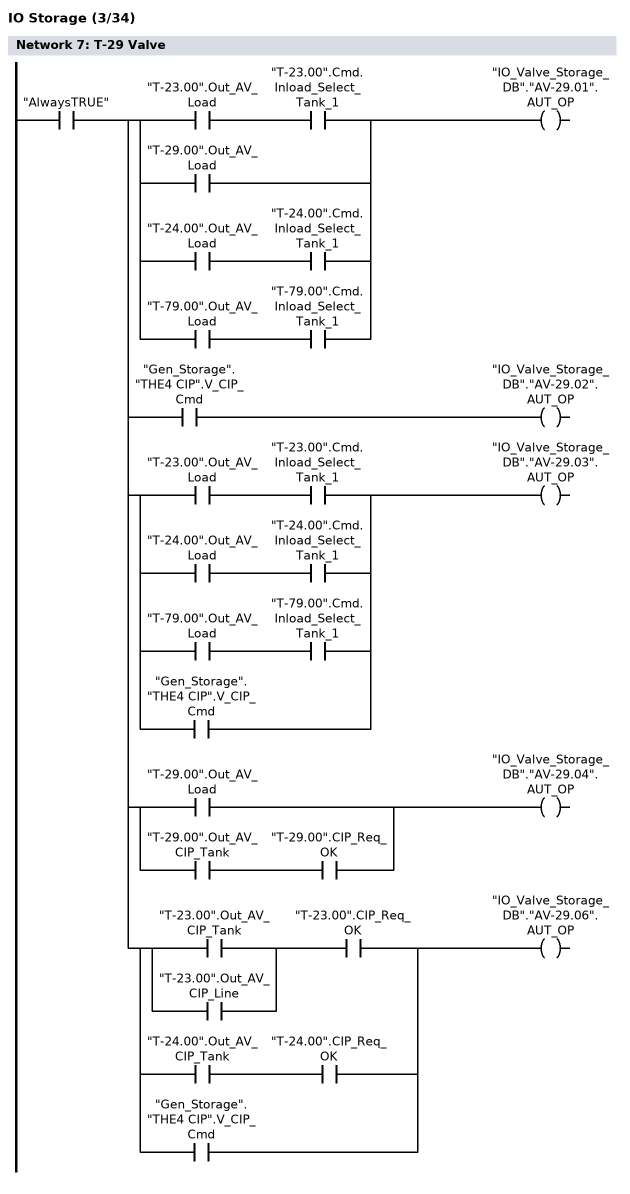
   RUNG wire#powerrail
      Contact( "AlwaysTRUE" )
      wire#w1
      Contact( "T-23.00".Out_AV_Load )
      Contact( "T-23.00".Cmd.Inload_Select_Tank_1 )
      wire#w2
      Coil( "IO_Valve_Storage_DB"."AV-29.01".AUT_OP )
   END_RUNG
   RUNG wire#w1
      Contact( "T-29.00".Out_AV_Load )
   END_RUNG wire#w2
   RUNG wire#w1
      Contact( "T-24.00".Out_AV_Load )
      Contact( "T-24.00".Cmd.Inload_Select_Tank_1 )
   END_RUNG wire#w2
   RUNG wire#w1
      Contact( "T-79.00".Out_AV_Load )
      Contact( "T-79.00".Cmd.Inload_Select_Tank_1 )
   END_RUNG wire#w2
   RUNG wire#w1
      Contact( "Gen_Storage"."THE4 CIP".V_CIP_Cmd )
      Coil( "IO_Valve_Storage_DB"."AV-29.02".AUT_OP )
   END_RUNG
   RUNG wire#w1
      Contact( "T-23.00".Out_AV_Load )
      Contact( "T-23.00".Cmd.Inload_Select_Tank_1 )
      wire#w3
      Coil( "IO_Valve_Storage_DB"."AV-29.03".AUT_OP )
   END_RUNG
   RUNG wire#w1
      Contact( "T-24.00".Out_AV_Load )
      Contact( "T-24.00".Cmd.Inload_Select_Tank_1 )
   END_RUNG wire#w3
   RUNG wire#w1
      Contact( "T-79.00".Out_AV_Load )
      Contact( "T-79.00".Cmd.Inload_Select_Tank_1 )
   END_RUNG wire#w3
   RUNG wire#w1
      Contact( "Gen_Storage"."THE4 CIP".V_CIP_Cmd )
   END_RUNG wire#w3
   RUNG wire#w1
      Contact( "T-29.00".Out_AV_Load )
      wire#w4
      Coil( "IO_Valve_Storage_DB"."AV-29.04".AUT_OP )
   END_RUNG
   RUNG wire#w1
      Contact( "T-29.00".Out_AV_CIP_Tank )
      Contact( "T-29.00".CIP_Req_OK )
   END_RUNG wire#w4
   RUNG wire#w1
      Contact( "T-23.00".Out_AV_CIP_Tank )
      wire#w5
      Contact( "T-23.00".CIP_Req_OK )
      wire#w6
      Coil( "IO_Valve_Storage_DB"."AV-29.06".AUT_OP )
   END_RUNG
   RUNG wire#w1
      Contact( "T-23.00".Out_AV_CIP_Line )
   END_RUNG wire#w5
   RUNG wire#w1
      Contact( "T-24.00".Out_AV_CIP_Tank )
      Contact( "T-24.00".CIP_Req_OK )
   END_RUNG wire#w6
   RUNG wire#w1
      Contact( "Gen_Storage"."THE4 CIP".V_CIP_Cmd )
   END_RUNG wire#w6
   // the same network as SCL:
   "IO_Valve_Storage_DB"."AV-29.01".AUT_OP := "AlwaysTRUE" AND (("T-23.00".Out_AV_Load AND "T-23.00".Cmd.Inload_Select_Tank_1) OR "T-29.00".Out_AV_Load OR ("T-24.00".Out_AV_Load AND "T-24.00".Cmd.Inload_Select_Tank_1) OR ("T-79.00".Out_AV_Load AND "T-79.00".Cmd.Inload_Select_Tank_1));
   "IO_Valve_Storage_DB"."AV-29.02".AUT_OP := "AlwaysTRUE" AND "Gen_Storage"."THE4 CIP".V_CIP_Cmd;
   "IO_Valve_Storage_DB"."AV-29.03".AUT_OP := "AlwaysTRUE" AND (("T-23.00".Out_AV_Load AND "T-23.00".Cmd.Inload_Select_Tank_1) OR ("T-24.00".Out_AV_Load AND "T-24.00".Cmd.Inload_Select_Tank_1) OR ("T-79.00".Out_AV_Load AND "T-79.00".Cmd.Inload_Select_Tank_1) OR "Gen_Storage"."THE4 CIP".V_CIP_Cmd);
   "IO_Valve_Storage_DB"."AV-29.04".AUT_OP := "AlwaysTRUE" AND ("T-29.00".Out_AV_Load OR ("T-29.00".Out_AV_CIP_Tank AND "T-29.00".CIP_Req_OK));
   "IO_Valve_Storage_DB"."AV-29.06".AUT_OP := "AlwaysTRUE" AND ((("T-23.00".Out_AV_CIP_Tank OR "T-23.00".Out_AV_CIP_Line) AND "T-23.00".CIP_Req_OK) OR ("T-24.00".Out_AV_CIP_Tank AND "T-24.00".CIP_Req_OK) OR "Gen_Storage"."THE4 CIP".V_CIP_Cmd);
END_REGION

REGION Network 9: T-23.00 ST-05
   // Inload 1 : THE-4
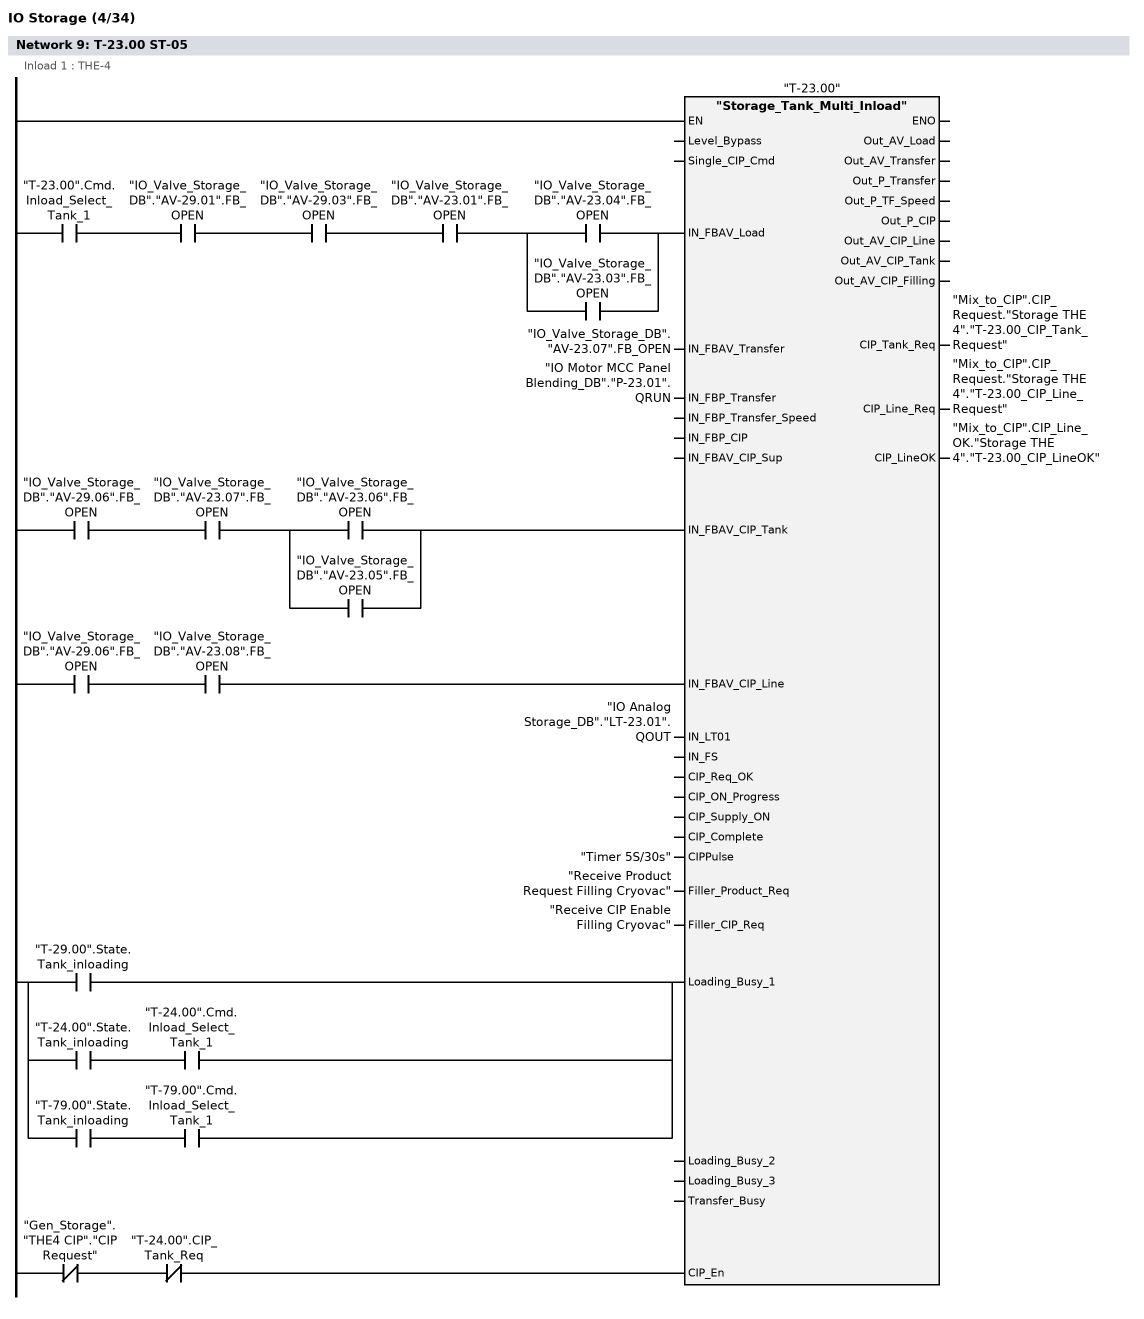
   RUNG wire#powerrail
      "T-23.00"(IN_FBAV_Load := wire#w2, IN_FBAV_CIP_Tank := wire#w4, IN_FBAV_CIP_Line := wire#w5, Loading_Busy_1 := wire#w6, CIP_En := wire#w7, Level_Bypass :=, Single_CIP_Cmd :=, IN_FBAV_Transfer := "IO_Valve_Storage_DB"."AV-23.07".FB_OPEN, IN_FBP_Transfer := "IO Motor MCC Panel Blending_DB"."P-23.01".QRUN, IN_FBP_Transfer_Speed :=, IN_FBP_CIP :=, IN_FBAV_CIP_Sup :=, IN_LT01 := "IO Analog Storage_DB"."LT-23.01".QOUT, IN_FS :=, CIP_Req_OK :=, CIP_ON_Progress :=, CIP_Supply_ON :=, CIP_Complete :=, CIPPulse := "Timer 5S/30s", Filler_Product_Req := "Receive Product Request Filling Cryovac", Filler_CIP_Req := "Receive CIP Enable Filling Cryovac", Loading_Busy_2 :=, Loading_Busy_3 :=, Transfer_Busy :=, Out_AV_Load =>, Out_AV_Transfer =>, Out_P_Transfer =>, Out_P_TF_Speed =>, Out_P_CIP =>, Out_AV_CIP_Line =>, Out_AV_CIP_Tank =>, Out_AV_CIP_Filling =>, CIP_Tank_Req => "Mix_to_CIP".CIP_Request."Storage THE 4"."T-23.00_CIP_Tank_Request", CIP_Line_Req => "Mix_to_CIP".CIP_Request."Storage THE 4"."T-23.00_CIP_Line_Request", CIP_LineOK => "Mix_to_CIP".CIP_Line_OK."Storage THE 4"."T-23.00_CIP_LineOK")
   END_RUNG
   RUNG wire#powerrail
      Contact( "T-23.00".Cmd.Inload_Select_Tank_1 )
      Contact( "IO_Valve_Storage_DB"."AV-29.01".FB_OPEN )
      Contact( "IO_Valve_Storage_DB"."AV-29.03".FB_OPEN )
      Contact( "IO_Valve_Storage_DB"."AV-23.01".FB_OPEN )
      wire#w1
      Contact( "IO_Valve_Storage_DB"."AV-23.04".FB_OPEN )
   END_RUNG wire#w2
   RUNG wire#w1
      Contact( "IO_Valve_Storage_DB"."AV-23.03".FB_OPEN )
   END_RUNG wire#w2
   RUNG wire#powerrail
      Contact( "IO_Valve_Storage_DB"."AV-29.06".FB_OPEN )
      Contact( "IO_Valve_Storage_DB"."AV-23.07".FB_OPEN )
      wire#w3
      Contact( "IO_Valve_Storage_DB"."AV-23.06".FB_OPEN )
   END_RUNG wire#w4
   RUNG wire#w3
      Contact( "IO_Valve_Storage_DB"."AV-23.05".FB_OPEN )
   END_RUNG wire#w4
   RUNG wire#powerrail
      Contact( "IO_Valve_Storage_DB"."AV-29.06".FB_OPEN )
      Contact( "IO_Valve_Storage_DB"."AV-23.08".FB_OPEN )
   END_RUNG wire#w5
   RUNG wire#powerrail
      Contact( "T-29.00".State.Tank_inloading )
   END_RUNG wire#w6
   RUNG wire#powerrail
      Contact( "T-24.00".State.Tank_inloading )
      Contact( "T-24.00".Cmd.Inload_Select_Tank_1 )
   END_RUNG wire#w6
   RUNG wire#powerrail
      Contact( "T-79.00".State.Tank_inloading )
      Contact( "T-79.00".Cmd.Inload_Select_Tank_1 )
   END_RUNG wire#w6
   RUNG wire#powerrail
      I_Contact( "Gen_Storage"."THE4 CIP"."CIP Request" )
      I_Contact( "T-24.00".CIP_Tank_Req )
   END_RUNG wire#w7
   // the same network as SCL:
   "T-23.00"(IN_FBAV_Load := "T-23.00".Cmd.Inload_Select_Tank_1 AND "IO_Valve_Storage_DB"."AV-29.01".FB_OPEN AND "IO_Valve_Storage_DB"."AV-29.03".FB_OPEN AND "IO_Valve_Storage_DB"."AV-23.01".FB_OPEN AND ("IO_Valve_Storage_DB"."AV-23.04".FB_OPEN OR "IO_Valve_Storage_DB"."AV-23.03".FB_OPEN),   // "Storage_Tank_Multi_Inload"
             IN_FBAV_Transfer := "IO_Valve_Storage_DB"."AV-23.07".FB_OPEN,
             IN_FBP_Transfer := "IO Motor MCC Panel Blending_DB"."P-23.01".QRUN,
             IN_FBAV_CIP_Tank := "IO_Valve_Storage_DB"."AV-29.06".FB_OPEN AND "IO_Valve_Storage_DB"."AV-23.07".FB_OPEN AND ("IO_Valve_Storage_DB"."AV-23.06".FB_OPEN OR "IO_Valve_Storage_DB"."AV-23.05".FB_OPEN),
             IN_FBAV_CIP_Line := "IO_Valve_Storage_DB"."AV-29.06".FB_OPEN AND "IO_Valve_Storage_DB"."AV-23.08".FB_OPEN,
             IN_LT01 := "IO Analog Storage_DB"."LT-23.01".QOUT,
             CIPPulse := "Timer 5S/30s",
             Filler_Product_Req := "Receive Product Request Filling Cryovac",
             Filler_CIP_Req := "Receive CIP Enable Filling Cryovac",
             Loading_Busy_1 := "T-29.00".State.Tank_inloading OR ("T-24.00".State.Tank_inloading AND "T-24.00".Cmd.Inload_Select_Tank_1) OR ("T-79.00".State.Tank_inloading AND "T-79.00".Cmd.Inload_Select_Tank_1),
             CIP_En := NOT "Gen_Storage"."THE4 CIP"."CIP Request" AND NOT "T-24.00".CIP_Tank_Req,
             CIP_Tank_Req => "Mix_to_CIP".CIP_Request."Storage THE 4"."T-23.00_CIP_Tank_Request",
             CIP_Line_Req => "Mix_to_CIP".CIP_Request."Storage THE 4"."T-23.00_CIP_Line_Request",
             CIP_LineOK => "Mix_to_CIP".CIP_Line_OK."Storage THE 4"."T-23.00_CIP_LineOK");
END_REGION

REGION Network 10: T-23 Valve
